LIN {X 0,Y 319.514,Z 305.497,A -85,B 0,C 180,E1 -15073.459,E2 -15073.459} C_VEL
LIN {X 0,Y 319.546,Z 305.495,A -85,B 0,C 180,E1 -15077.015,E2 -15077.015} C_VEL
LIN {X 0,Y 319.525,Z 305.485,A -85,B 0,C 180,E1 -15080.367,E2 -15080.367} C_VEL
LIN {X 0,Y 319.573,Z 305.485,A -85,B 0,C 180,E1 -15084.457,E2 -15084.457} C_VEL
LIN {X 0,Y 319.518,Z 305.495,A -85,B 0,C 180,E1 -15088.137,E2 -15088.137} C_VEL
LIN {X 0,Y 319.563,Z 305.487,A -85,B 0,C 180,E1 -15091.604,E2 -15091.604} C_VEL
LIN {X 0,Y 319.519,Z 305.494,A -85,B 0,C 180,E1 -15095.297,E2 -15095.297} C_VEL
LIN {X 0,Y 319.555,Z 305.486,A -85,B 0,C 180,E1 -15098.045,E2 -15098.045} C_VEL
LIN {X 0,Y 319.579,Z 305.489,A -85,B 0,C 180,E1 -15102.068,E2 -15102.068} C_VEL
LIN {X 0,Y 319.702,Z 305.469,A -85,B 0,C 180,E1 -15106.006,E2 -15106.006} C_VEL
LIN {X 0,Y 319.728,Z 305.469,A -85,B 0,C 180,E1 -15109.872,E2 -15109.872} C_VEL
LIN {X 0,Y 319.89,Z 305.447,A -85,B 0,C 180,E1 -15113.693,E2 -15113.693} C_VEL
LIN {X 0,Y 319.945,Z 305.439,A -85,B 0,C 180,E1 -15117.482,E2 -15117.482} C_VEL
LIN {X 0,Y 319.988,Z 305.436,A -85,B 0,C 180,E1 -15121.258,E2 -15121.258} C_VEL
LIN {X 0,Y 319.705,Z 305.464,A -85,B 0,C 180,E1 -15125.044,E2 -15125.044} C_VEL
LIN {X 0,Y 319.844,Z 305.454,A -85,B 0,C 180,E1 -15127.576,E2 -15127.576} C_VEL
LIN {X 0,Y 319.702,Z 305.473,A -85,B 0,C 180,E1 -15131.411,E2 -15131.411} C_VEL
LIN {X 0,Y 319.656,Z 305.473,A -85,B 0,C 180,E1 -15134.677,E2 -15134.677} C_VEL
LIN {X 0,Y 319.579,Z 305.489,A -85,B 0,C 180,E1 -15137.931,E2 -15137.931} C_VEL
LIN {X 0,Y 319.555,Z 305.486,A -85,B 0,C 180,E1 -15141.955,E2 -15141.955} C_VEL
LIN {X 0,Y 319.542,Z 305.492,A -85,B 0,C 180,E1 -15146.096,E2 -15146.096} C_VEL
LIN {X 0,Y 319.534,Z 305.493,A -85,B 0,C 180,E1 -15148.939,E2 -15148.939} C_VEL
LIN {X 0,Y 319.517,Z 305.495,A -85,B 0,C 180,E1 -15151.863,E2 -15151.863} C_VEL
LIN {X 0,Y 319.572,Z 305.486,A -85,B 0,C 180,E1 -15155.543,E2 -15155.543} C_VEL
LIN {X 0,Y 319.523,Z 305.485,A -85,B 0,C 180,E1 -15159.663,E2 -15159.663} C_VEL
LIN {X 0,Y 319.513,Z 305.496,A -85,B 0,C 180,E1 -15163.46,E2 -15163.46} C_VEL
LIN {X 0,Y 319.545,Z 305.488,A -85,B 0,C 180,E1 -15167.016,E2 -15167.016} C_VEL
LIN {X 0,Y 319.541,Z 305.489,A -85,B 0,C 180,E1 -15170.371,E2 -15170.371} C_VEL
LIN {X 0,Y 319.576,Z 305.488,A -85,B 0,C 180,E1 -15174.458,E2 -15174.458} C_VEL
LIN {X 0,Y 319.521,Z 305.497,A -85,B 0,C 180,E1 -15178.138,E2 -15178.138} C_VEL
LIN {X 0,Y 319.566,Z 305.489,A -85,B 0,C 180,E1 -15181.605,E2 -15181.605} C_VEL
LIN {X 0,Y 319.634,Z 305.687,A -85,B 0,C 180,E1 -15183.913,E2 -15183.913} C_VEL
LIN {X 0,Y 321.119,Z 313.482,A -85,B 0,C 180,E1 -15186.811,E2 -15186.811} C_VEL
LIN {X 0,Y 321.518,Z 317.355,A -85,B 0,C 180,E1 -15188.186,E2 -15188.186} C_VEL
LIN {X 0,Y 321.084,Z 323.649,A -85,B 0,C 180,E1 -15190.254,E2 -15190.254} C_VEL
LIN {X 0,Y 321.598,Z 327,A -85,B 0,C 180,E1 -15190.437,E2 -15190.437} C_VEL
LIN {X 0,Y 325.831,Z 351.509,A -85,B 0,C 180,E1 -15191.261,E2 -15191.261} C_VEL
LIN {X 0,Y 325.681,Z 374.115,A -85,B 0,C 180,E1 -15191.767,E2 -15191.767} C_VEL
LIN {X 0,Y 325.184,Z 400.782,A -85,B 0,C 180,E1 -15192.388,E2 -15192.388} C_VEL
LIN {X 0,Y 324.681,Z 411.953,A -85,B 0,C 180,E1 -15192.847,E2 -15192.847} C_VEL
LIN {X 0,Y 323.933,Z 423.638,A -85,B 0,C 180,E1 -15193.618,E2 -15193.618} C_VEL
LIN {X 0,Y 323.143,Z 432.319,A -85,B 0,C 180,E1 -15194.387,E2 -15194.387} C_VEL
LIN {X 0,Y 322.282,Z 440.61,A -85,B 0,C 180,E1 -15195.315,E2 -15195.315} C_VEL
LIN {X 0,Y 321.43,Z 448.456,A -85,B 0,C 180,E1 -15196.406,E2 -15196.406} C_VEL
LIN {X 0,Y 320.573,Z 455.792,A -85,B 0,C 180,E1 -15197.658,E2 -15197.658} C_VEL
LIN {X 0,Y 319.668,Z 463.231,A -85,B 0,C 180,E1 -15199.23,E2 -15199.23} C_VEL
LIN {X 0,Y 318.847,Z 470.019,A -85,B 0,C 180,E1 -15201.124,E2 -15201.124} C_VEL
LIN {X 0,Y 318.301,Z 475.173,A -85,B 0,C 180,E1 -15203.025,E2 -15203.025} C_VEL
LIN {X 0,Y 318.001,Z 478.956,A -85,B 0,C 180,E1 -15204.928,E2 -15204.928} C_VEL
LIN {X 0,Y 317.894,Z 480.692,A -85,B 0,C 180,E1 -15206.197,E2 -15206.197} C_VEL
LIN {X 0,Y 317.77,Z 481.935,A -85,B 0,C 180,E1 -15207.465,E2 -15207.465} C_VEL
LIN {X 0,Y 317.7,Z 482.708,A -85,B 0,C 180,E1 -15208.732,E2 -15208.732} C_VEL
LIN {X 0,Y 317.677,Z 483,A -85,B 0,C 180,E1 -15210,E2 -15210} C_VEL
LIN {X 0,Y 317.7,Z 482.703,A -85,B 0,C 180,E1 -15211.268,E2 -15211.268} C_VEL
LIN {X 0,Y 317.77,Z 481.92,A -85,B 0,C 180,E1 -15212.535,E2 -15212.535} C_VEL
LIN {X 0,Y 317.893,Z 480.666,A -85,B 0,C 180,E1 -15213.803,E2 -15213.803} C_VEL
LIN {X 0,Y 318.041,Z 477.844,A -85,B 0,C 180,E1 -15215.665,E2 -15215.665} C_VEL
LIN {X 0,Y 318.312,Z 475.126,A -85,B 0,C 180,E1 -15216.975,E2 -15216.975} C_VEL
LIN {X 0,Y 318.846,Z 469.956,A -85,B 0,C 180,E1 -15218.876,E2 -15218.876} C_VEL
LIN {X 0,Y 319.665,Z 463.14,A -85,B 0,C 180,E1 -15220.77,E2 -15220.77} C_VEL
LIN {X 0,Y 320.563,Z 455.687,A -85,B 0,C 180,E1 -15222.342,E2 -15222.342} C_VEL
LIN {X 0,Y 321.411,Z 448.334,A -85,B 0,C 180,E1 -15223.595,E2 -15223.595} C_VEL
LIN {X 0,Y 322.279,Z 440.457,A -85,B 0,C 180,E1 -15224.685,E2 -15224.685} C_VEL
LIN {X 0,Y 323.17,Z 432.129,A -85,B 0,C 180,E1 -15225.612,E2 -15225.612} C_VEL
LIN {X 0,Y 324.041,Z 421.482,A -85,B 0,C 180,E1 -15226.538,E2 -15226.538} C_VEL
LIN {X 0,Y 324.762,Z 409.87,A -85,B 0,C 180,E1 -15227.229,E2 -15227.229} C_VEL
LIN {X 0,Y 325.152,Z 401.415,A -85,B 0,C 180,E1 -15227.573,E2 -15227.573} C_VEL
LIN {X 0,Y 325.626,Z 375.19,A -85,B 0,C 180,E1 -15228.191,E2 -15228.191} C_VEL
LIN {X 0,Y 325.9,Z 352.19,A -85,B 0,C 180,E1 -15228.698,E2 -15228.698} C_VEL
LIN {X 0,Y 321.555,Z 326.797,A -85,B 0,C 180,E1 -15229.548,E2 -15229.548} C_VEL
LIN {X 0,Y 321.053,Z 323.814,A -85,B 0,C 180,E1 -15229.701,E2 -15229.701} C_VEL
LIN {X 0,Y 321.433,Z 319.241,A -85,B 0,C 180,E1 -15231.147,E2 -15231.147} C_VEL
LIN {X 0,Y 321.373,Z 315.374,A -85,B 0,C 180,E1 -15232.487,E2 -15232.487} C_VEL
LIN {X 0,Y 319.816,Z 306.575,A -85,B 0,C 180,E1 -15235.713,E2 -15235.713} C_VEL
LIN {X 0,Y 319.63,Z 305.559,A -85,B 0,C 180,E1 -15236.176,E2 -15236.176} C_VEL
LIN {X 0,Y 319.557,Z 305.488,A -85,B 0,C 180,E1 -15240.386,E2 -15240.386} C_VEL
LIN {X 0,Y 319.574,Z 305.491,A -85,B 0,C 180,E1 -15243.352,E2 -15243.352} C_VEL
LIN {X 0,Y 319.552,Z 305.489,A -85,B 0,C 180,E1 -15246.427,E2 -15246.427} C_VEL
LIN {X 0,Y 319.524,Z 305.491,A -85,B 0,C 180,E1 -15249.661,E2 -15249.661} C_VEL
LIN {X 0,Y 319.513,Z 305.497,A -85,B 0,C 180,E1 -15253.459,E2 -15253.459} C_VEL
LIN {X 0,Y 319.544,Z 305.495,A -85,B 0,C 180,E1 -15257.015,E2 -15257.015} C_VEL
LIN {X 0,Y 319.509,Z 305.486,A -85,B 0,C 180,E1 -15260.365,E2 -15260.365} C_VEL
LIN {X 0,Y 319.572,Z 305.486,A -85,B 0,C 180,E1 -15264.457,E2 -15264.457} C_VEL
LIN {X 0,Y 319.517,Z 305.495,A -85,B 0,C 180,E1 -15268.137,E2 -15268.137} C_VEL
LIN {X 0,Y 319.562,Z 305.487,A -85,B 0,C 180,E1 -15271.604,E2 -15271.604} C_VEL
LIN {X 0,Y 319.518,Z 305.494,A -85,B 0,C 180,E1 -15275.297,E2 -15275.297} C_VEL
LIN {X 0,Y 319.555,Z 305.486,A -85,B 0,C 180,E1 -15278.045,E2 -15278.045} C_VEL
LIN {X 0,Y 319.578,Z 305.489,A -85,B 0,C 180,E1 -15282.069,E2 -15282.069} C_VEL
LIN {X 0,Y 319.702,Z 305.469,A -85,B 0,C 180,E1 -15286.007,E2 -15286.007} C_VEL
LIN {X 0,Y 319.727,Z 305.469,A -85,B 0,C 180,E1 -15289.872,E2 -15289.872} C_VEL
LIN {X 0,Y 319.89,Z 305.447,A -85,B 0,C 180,E1 -15293.693,E2 -15293.693} C_VEL
LIN {X 0,Y 319.945,Z 305.439,A -85,B 0,C 180,E1 -15297.482,E2 -15297.482} C_VEL
LIN {X 0,Y 319.988,Z 305.436,A -85,B 0,C 180,E1 -15301.259,E2 -15301.259} C_VEL
LIN {X 0,Y 319.706,Z 305.464,A -85,B 0,C 180,E1 -15305.045,E2 -15305.045} C_VEL
LIN {X 0,Y 319.844,Z 305.454,A -85,B 0,C 180,E1 -15307.576,E2 -15307.576} C_VEL
LIN {X 0,Y 319.702,Z 305.473,A -85,B 0,C 180,E1 -15311.411,E2 -15311.411} C_VEL
LIN {X 0,Y 319.656,Z 305.473,A -85,B 0,C 180,E1 -15314.678,E2 -15314.678} C_VEL
LIN {X 0,Y 319.579,Z 305.489,A -85,B 0,C 180,E1 -15317.932,E2 -15317.932} C_VEL
LIN {X 0,Y 319.555,Z 305.486,A -85,B 0,C 180,E1 -15321.955,E2 -15321.955} C_VEL
LIN {X 0,Y 319.542,Z 305.492,A -85,B 0,C 180,E1 -15326.096,E2 -15326.096} C_VEL
LIN {X 0,Y 319.534,Z 305.493,A -85,B 0,C 180,E1 -15328.939,E2 -15328.939} C_VEL
LIN {X 0,Y 319.518,Z 305.495,A -85,B 0,C 180,E1 -15331.864,E2 -15331.864} C_VEL
LIN {X 0,Y 319.572,Z 305.486,A -85,B 0,C 180,E1 -15335.543,E2 -15335.543} C_VEL
LIN {X 0,Y 319.524,Z 305.484,A -85,B 0,C 180,E1 -15339.663,E2 -15339.663} C_VEL
LIN {X 0,Y 319.514,Z 305.496,A -85,B 0,C 180,E1 -15343.461,E2 -15343.461} C_VEL
LIN {X 0,Y 319.546,Z 305.489,A -85,B 0,C 180,E1 -15347.016,E2 -15347.016} C_VEL
LIN {X 0,Y 319.542,Z 305.488,A -85,B 0,C 180,E1 -15350.371,E2 -15350.371} C_VEL
LIN {X 0,Y 319.577,Z 305.488,A -85,B 0,C 180,E1 -15354.458,E2 -15354.458} C_VEL
LIN {X 0,Y 319.522,Z 305.496,A -85,B 0,C 180,E1 -15358.138,E2 -15358.138} C_VEL
LIN {X 0,Y 319.542,Z 305.493,A -85,B 0,C 180,E1 -15361.614,E2 -15361.614} C_VEL
LIN {X 0,Y 319.63,Z 305.684,A -85,B 0,C 180,E1 -15363.98,E2 -15363.98} C_VEL
LIN {X 0,Y 321.085,Z 313.335,A -85,B 0,C 180,E1 -15366.825,E2 -15366.825} C_VEL
LIN {X 0,Y 321.51,Z 317.158,A -85,B 0,C 180,E1 -15368.186,E2 -15368.186} C_VEL
LIN {X 0,Y 321.053,Z 323.63,A -85,B 0,C 180,E1 -15370.308,E2 -15370.308} C_VEL
LIN {X 0,Y 321.428,Z 326.151,A -85,B 0,C 180,E1 -15370.474,E2 -15370.474} C_VEL
LIN {X 0,Y 325.861,Z 352.125,A -85,B 0,C 180,E1 -15371.343,E2 -15371.343} C_VEL
LIN {X 0,Y 325.2,Z 399.977,A -85,B 0,C 180,E1 -15372.43,E2 -15372.43} C_VEL
LIN {X 0,Y 324.814,Z 408.948,A -85,B 0,C 180,E1 -15372.774,E2 -15372.774} C_VEL
LIN {X 0,Y 324.273,Z 418.484,A -85,B 0,C 180,E1 -15373.312,E2 -15373.312} C_VEL
LIN {X 0,Y 323.521,Z 428.497,A -85,B 0,C 180,E1 -15374.083,E2 -15374.083} C_VEL
LIN {X 0,Y 322.486,Z 438.884,A -85,B 0,C 180,E1 -15375.163,E2 -15375.163} C_VEL
LIN {X 0,Y 321.565,Z 447.028,A -85,B 0,C 180,E1 -15376.251,E2 -15376.251} C_VEL
LIN {X 0,Y 320.834,Z 453.747,A -85,B 0,C 180,E1 -15377.347,E2 -15377.347} C_VEL
LIN {X 0,Y 320.021,Z 460.112,A -85,B 0,C 180,E1 -15378.601,E2 -15378.601} C_VEL
LIN {X 0,Y 319.24,Z 466.576,A -85,B 0,C 180,E1 -15380.177,E2 -15380.177} C_VEL
LIN {X 0,Y 318.679,Z 471.734,A -85,B 0,C 180,E1 -15381.759,E2 -15381.759} C_VEL
LIN {X 0,Y 318.157,Z 476.676,A -85,B 0,C 180,E1 -15383.741,E2 -15383.741} C_VEL
LIN {X 0,Y 318.009,Z 478.838,A -85,B 0,C 180,E1 -15384.929,E2 -15384.929} C_VEL
LIN {X 0,Y 317.899,Z 480.609,A -85,B 0,C 180,E1 -15386.197,E2 -15386.197} C_VEL
LIN {X 0,Y 317.772,Z 481.886,A -85,B 0,C 180,E1 -15387.465,E2 -15387.465} C_VEL
LIN {X 0,Y 317.701,Z 482.691,A -85,B 0,C 180,E1 -15388.732,E2 -15388.732} C_VEL
LIN {X 0,Y 317.679,Z 482.998,A -85,B 0,C 180,E1 -15390,E2 -15390} C_VEL
LIN {X 0,Y 317.697,Z 482.719,A -85,B 0,C 180,E1 -15391.268,E2 -15391.268} C_VEL
LIN {X 0,Y 317.76,Z 481.97,A -85,B 0,C 180,E1 -15392.535,E2 -15392.535} C_VEL
LIN {X 0,Y 317.87,Z 480.75,A -85,B 0,C 180,E1 -15393.803,E2 -15393.803} C_VEL
LIN {X 0,Y 318.029,Z 478.009,A -85,B 0,C 180,E1 -15395.639,E2 -15395.639} C_VEL
LIN {X 0,Y 318.309,Z 475.28,A -85,B 0,C 180,E1 -15396.975,E2 -15396.975} C_VEL
LIN {X 0,Y 318.839,Z 470.153,A -85,B 0,C 180,E1 -15398.876,E2 -15398.876} C_VEL
LIN {X 0,Y 319.502,Z 464.639,A -85,B 0,C 180,E1 -15400.455,E2 -15400.455} C_VEL
LIN {X 0,Y 320.377,Z 457.713,A -85,B 0,C 180,E1 -15402.028,E2 -15402.028} C_VEL
LIN {X 0,Y 321.284,Z 449.762,A -85,B 0,C 180,E1 -15403.439,E2 -15403.439} C_VEL
LIN {X 0,Y 322.108,Z 442.181,A -85,B 0,C 180,E1 -15404.531,E2 -15404.531} C_VEL
LIN {X 0,Y 323.005,Z 434.237,A -85,B 0,C 180,E1 -15405.458,E2 -15405.458} C_VEL
LIN {X 0,Y 323.747,Z 426.031,A -85,B 0,C 180,E1 -15406.23,E2 -15406.23} C_VEL
LIN {X 0,Y 324.389,Z 417.714,A -85,B 0,C 180,E1 -15406.844,E2 -15406.844} C_VEL
LIN {X 0,Y 324.828,Z 408.722,A -85,B 0,C 180,E1 -15407.347,E2 -15407.347} C_VEL
LIN {X 0,Y 325.258,Z 399.317,A -85,B 0,C 180,E1 -15407.699,E2 -15407.699} C_VEL
LIN {X 0,Y 325.92,Z 352.078,A -85,B 0,C 180,E1 -15408.765,E2 -15408.765} C_VEL
LIN {X 0,Y 321.836,Z 328.161,A -85,B 0,C 180,E1 -15409.566,E2 -15409.566} C_VEL
LIN {X 0,Y 321.058,Z 323.761,A -85,B 0,C 180,E1 -15409.776,E2 -15409.776} C_VEL
LIN {X 0,Y 321.492,Z 317.485,A -85,B 0,C 180,E1 -15411.816,E2 -15411.816} C_VEL
LIN {X 0,Y 320.766,Z 311.628,A -85,B 0,C 180,E1 -15413.912,E2 -15413.912} C_VEL
LIN {X 0,Y 319.606,Z 305.566,A -85,B 0,C 180,E1 -15416.222,E2 -15416.222} C_VEL
LIN {X 0,Y 319.541,Z 305.493,A -85,B 0,C 180,E1 -15418.938,E2 -15418.938} C_VEL
LIN {X 0,Y 319.522,Z 305.497,A -85,B 0,C 180,E1 -15421.862,E2 -15421.862} C_VEL
LIN {X 0,Y 319.577,Z 305.487,A -85,B 0,C 180,E1 -15425.542,E2 -15425.542} C_VEL
LIN {X 0,Y 319.525,Z 305.491,A -85,B 0,C 180,E1 -15429.661,E2 -15429.661} C_VEL
LIN {X 0,Y 319.491,Z 305.492,A -85,B 0,C 180,E1 -15431.235,E2 -15431.235} C_VEL
LIN {X 0,Y 318.864,Z 305.576,A -85,B 0,C 180,E1 -15432.287,E2 -15432.287} C_VEL
LIN {X 0,Y 316.003,Z 305.934,A -85,B 0,C 180,E1 -15433.997,E2 -15433.997} C_VEL
LIN {X 0,Y 313.554,Z 306.241,A -85,B 0,C 180,E1 -15435.383,E2 -15435.383} C_VEL
LIN {X 0,Y 312.509,Z 306.368,A -85,B 0,C 180,E1 -15436.458,E2 -15436.458} C_VEL
LIN {X 0,Y 312.429,Z 306.374,A -85,B 0,C 180,E1 -15436.822,E2 -15436.822} C_VEL
LIN {X 0,Y 312.46,Z 306.361,A -85,B 0,C 180,E1 -15440.965,E2 -15440.965} C_VEL
LIN {X 0,Y 312.524,Z 306.362,A -85,B 0,C 180,E1 -15444.219,E2 -15444.219} C_VEL
LIN {X 0,Y 312.496,Z 306.37,A -85,B 0,C 180,E1 -15447.333,E2 -15447.333} C_VEL
LIN {X 0,Y 312.498,Z 306.368,A -85,B 0,C 180,E1 -15451.292,E2 -15451.292} C_VEL
LIN {X 0,Y 312.51,Z 306.371,A -85,B 0,C 180,E1 -15454.704,E2 -15454.704} C_VEL
LIN {X 0,Y 312.532,Z 306.359,A -85,B 0,C 180,E1 -15457.525,E2 -15457.525} C_VEL
LIN {X 0,Y 312.539,Z 306.364,A -85,B 0,C 180,E1 -15461.65,E2 -15461.65} C_VEL
LIN {X 0,Y 312.644,Z 306.346,A -85,B 0,C 180,E1 -15465.684,E2 -15465.684} C_VEL
LIN {X 0,Y 312.678,Z 306.346,A -85,B 0,C 180,E1 -15469.641,E2 -15469.641} C_VEL
LIN {X 0,Y 312.788,Z 306.335,A -85,B 0,C 180,E1 -15472.252,E2 -15472.252} C_VEL
LIN {X 0,Y 312.677,Z 306.339,A -85,B 0,C 180,E1 -15474.842,E2 -15474.842} C_VEL
LIN {X 0,Y 312.957,Z 306.312,A -85,B 0,C 180,E1 -15478.713,E2 -15478.713} C_VEL
LIN {X 0,Y 312.956,Z 306.312,A -85,B 0,C 180,E1 -15481.287,E2 -15481.287} C_VEL
LIN {X 0,Y 312.832,Z 306.326,A -85,B 0,C 180,E1 -15486.449,E2 -15486.449} C_VEL
LIN {X 0,Y 312.675,Z 306.346,A -85,B 0,C 180,E1 -15490.359,E2 -15490.359} C_VEL
LIN {X 0,Y 312.643,Z 306.346,A -85,B 0,C 180,E1 -15494.316,E2 -15494.316} C_VEL
LIN {X 0,Y 312.539,Z 306.364,A -85,B 0,C 180,E1 -15498.35,E2 -15498.35} C_VEL
LIN {X 0,Y 312.531,Z 306.359,A -85,B 0,C 180,E1 -15502.475,E2 -15502.475} C_VEL
LIN {X 0,Y 312.5,Z 306.37,A -85,B 0,C 180,E1 -15505.899,E2 -15505.899} C_VEL
LIN {X 0,Y 312.488,Z 306.368,A -85,B 0,C 180,E1 -15509.656,E2 -15509.656} C_VEL
LIN {X 0,Y 312.513,Z 306.368,A -85,B 0,C 180,E1 -15513.689,E2 -15513.689} C_VEL
LIN {X 0,Y 312.503,Z 306.359,A -85,B 0,C 180,E1 -15517.388,E2 -15517.388} C_VEL
LIN {X 0,Y 312.435,Z 306.368,A -85,B 0,C 180,E1 -15520.718,E2 -15520.718} C_VEL
LIN {X 0,Y 312.444,Z 306.376,A -85,B 0,C 180,E1 -15524.211,E2 -15524.211} C_VEL
LIN {X 0,Y 312.448,Z 306.367,A -85,B 0,C 180,E1 -15527.926,E2 -15527.926} C_VEL
LIN {X 0,Y 312.479,Z 306.372,A -85,B 0,C 180,E1 -15531.923,E2 -15531.923} C_VEL
LIN {X 0,Y 312.527,Z 306.366,A -85,B 0,C 180,E1 -15534.221,E2 -15534.221} C_VEL
LIN {X 0,Y 312.498,Z 306.37,A -85,B 0,C 180,E1 -15537.334,E2 -15537.334} C_VEL
LIN {X 0,Y 312.502,Z 306.369,A -85,B 0,C 180,E1 -15541.293,E2 -15541.293} C_VEL
LIN {X 0,Y 312.588,Z 306.579,A -85,B 0,C 180,E1 -15543.61,E2 -15543.61} C_VEL
LIN {X 0,Y 314.303,Z 315.843,A -85,B 0,C 180,E1 -15547.121,E2 -15547.121} C_VEL
LIN {X 0,Y 314.384,Z 321.26,A -85,B 0,C 180,E1 -15549.043,E2 -15549.043} C_VEL
LIN {X 0,Y 314.178,Z 323.787,A -85,B 0,C 180,E1 -15549.822,E2 -15549.822} C_VEL
LIN {X 0,Y 315.376,Z 330.306,A -85,B 0,C 180,E1 -15550.113,E2 -15550.113} C_VEL
LIN {X 0,Y 319.287,Z 353.525,A -85,B 0,C 180,E1 -15550.909,E2 -15550.909} C_VEL
LIN {X 0,Y 318.496,Z 399.599,A -85,B 0,C 180,E1 -15551.967,E2 -15551.967} C_VEL
LIN {X 0,Y 318.075,Z 408.641,A -85,B 0,C 180,E1 -15552.314,E2 -15552.314} C_VEL
LIN {X 0,Y 317.489,Z 418.259,A -85,B 0,C 180,E1 -15552.862,E2 -15552.862} C_VEL
LIN {X 0,Y 316.805,Z 427.389,A -85,B 0,C 180,E1 -15553.57,E2 -15553.57} C_VEL
LIN {X 0,Y 315.736,Z 438.154,A -85,B 0,C 180,E1 -15554.673,E2 -15554.673} C_VEL
LIN {X 0,Y 314.752,Z 446.418,A -85,B 0,C 180,E1 -15555.782,E2 -15555.782} C_VEL
LIN {X 0,Y 313.854,Z 454.091,A -85,B 0,C 180,E1 -15557.061,E2 -15557.061} C_VEL
LIN {X 0,Y 313.039,Z 460.404,A -85,B 0,C 180,E1 -15558.343,E2 -15558.343} C_VEL
LIN {X 0,Y 312.335,Z 465.648,A -85,B 0,C 180,E1 -15559.63,E2 -15559.63} C_VEL
LIN {X 0,Y 311.818,Z 470.02,A -85,B 0,C 180,E1 -15560.923,E2 -15560.923} C_VEL
LIN {X 0,Y 311.246,Z 475.174,A -85,B 0,C 180,E1 -15562.866,E2 -15562.866} C_VEL
LIN {X 0,Y 310.916,Z 478.956,A -85,B 0,C 180,E1 -15564.813,E2 -15564.813} C_VEL
LIN {X 0,Y 310.809,Z 480.693,A -85,B 0,C 180,E1 -15566.11,E2 -15566.11} C_VEL
LIN {X 0,Y 310.696,Z 481.936,A -85,B 0,C 180,E1 -15567.407,E2 -15567.407} C_VEL
LIN {X 0,Y 310.617,Z 482.708,A -85,B 0,C 180,E1 -15568.704,E2 -15568.704} C_VEL
LIN {X 0,Y 310.592,Z 483,A -85,B 0,C 180,E1 -15570,E2 -15570} C_VEL
LIN {X 0,Y 310.617,Z 482.703,A -85,B 0,C 180,E1 -15571.296,E2 -15571.296} C_VEL
LIN {X 0,Y 310.696,Z 481.92,A -85,B 0,C 180,E1 -15572.593,E2 -15572.593} C_VEL
LIN {X 0,Y 310.808,Z 480.666,A -85,B 0,C 180,E1 -15573.89,E2 -15573.89} C_VEL
LIN {X 0,Y 310.912,Z 478.918,A -85,B 0,C 180,E1 -15575.188,E2 -15575.188} C_VEL
LIN {X 0,Y 311.251,Z 475.125,A -85,B 0,C 180,E1 -15577.134,E2 -15577.134} C_VEL
LIN {X 0,Y 311.817,Z 469.955,A -85,B 0,C 180,E1 -15579.077,E2 -15579.077} C_VEL
LIN {X 0,Y 312.667,Z 463.138,A -85,B 0,C 180,E1 -15581.014,E2 -15581.014} C_VEL
LIN {X 0,Y 313.64,Z 455.684,A -85,B 0,C 180,E1 -15582.619,E2 -15582.619} C_VEL
LIN {X 0,Y 314.501,Z 448.331,A -85,B 0,C 180,E1 -15583.899,E2 -15583.899} C_VEL
LIN {X 0,Y 315.434,Z 440.453,A -85,B 0,C 180,E1 -15585.011,E2 -15585.011} C_VEL
LIN {X 0,Y 316.354,Z 432.124,A -85,B 0,C 180,E1 -15585.957,E2 -15585.957} C_VEL
LIN {X 0,Y 317.24,Z 421.476,A -85,B 0,C 180,E1 -15586.903,E2 -15586.903} C_VEL
LIN {X 0,Y 318.004,Z 409.861,A -85,B 0,C 180,E1 -15587.607,E2 -15587.607} C_VEL
LIN {X 0,Y 318.41,Z 401.4,A -85,B 0,C 180,E1 -15587.958,E2 -15587.958} C_VEL
LIN {X 0,Y 318.889,Z 375.169,A -85,B 0,C 180,E1 -15588.589,E2 -15588.589} C_VEL
LIN {X 0,Y 319.191,Z 353.155,A -85,B 0,C 180,E1 -15589.083,E2 -15589.083} C_VEL
LIN {X 0,Y 314.775,Z 327.23,A -85,B 0,C 180,E1 -15589.976,E2 -15589.976} C_VEL
LIN {X 0,Y 314.159,Z 323.735,A -85,B 0,C 180,E1 -15590.165,E2 -15590.165} C_VEL
LIN {X 0,Y 314.491,Z 319.239,A -85,B 0,C 180,E1 -15591.637,E2 -15591.637} C_VEL
LIN {X 0,Y 314.047,Z 314.28,A -85,B 0,C 180,E1 -15593.432,E2 -15593.432} C_VEL
LIN {X 0,Y 312.57,Z 306.452,A -85,B 0,C 180,E1 -15596.446,E2 -15596.446} C_VEL
LIN {X 0,Y 312.493,Z 306.372,A -85,B 0,C 180,E1 -15599.655,E2 -15599.655} C_VEL
LIN {X 0,Y 312.517,Z 306.366,A -85,B 0,C 180,E1 -15603.688,E2 -15603.688} C_VEL
LIN {X 0,Y 312.51,Z 306.372,A -85,B 0,C 180,E1 -15607.386,E2 -15607.386} C_VEL
LIN {X 0,Y 312.435,Z 306.372,A -85,B 0,C 180,E1 -15610.717,E2 -15610.717} C_VEL
LIN {X 0,Y 312.445,Z 306.374,A -85,B 0,C 180,E1 -15614.21,E2 -15614.21} C_VEL
LIN {X 0,Y 312.448,Z 306.372,A -85,B 0,C 180,E1 -15617.925,E2 -15617.925} C_VEL
LIN {X 0,Y 312.469,Z 306.361,A -85,B 0,C 180,E1 -15621.924,E2 -15621.924} C_VEL
LIN {X 0,Y 312.523,Z 306.362,A -85,B 0,C 180,E1 -15624.219,E2 -15624.219} C_VEL
LIN {X 0,Y 312.495,Z 306.37,A -85,B 0,C 180,E1 -15627.333,E2 -15627.333} C_VEL
LIN {X 0,Y 312.498,Z 306.368,A -85,B 0,C 180,E1 -15631.292,E2 -15631.292} C_VEL
LIN {X 0,Y 312.509,Z 306.371,A -85,B 0,C 180,E1 -15634.704,E2 -15634.704} C_VEL
LIN {X 0,Y 312.531,Z 306.359,A -85,B 0,C 180,E1 -15637.525,E2 -15637.525} C_VEL
LIN {X 0,Y 312.539,Z 306.364,A -85,B 0,C 180,E1 -15641.65,E2 -15641.65} C_VEL
LIN {X 0,Y 312.644,Z 306.346,A -85,B 0,C 180,E1 -15645.684,E2 -15645.684} C_VEL
LIN {X 0,Y 312.677,Z 306.346,A -85,B 0,C 180,E1 -15649.641,E2 -15649.641} C_VEL
LIN {X 0,Y 312.788,Z 306.335,A -85,B 0,C 180,E1 -15652.252,E2 -15652.252} C_VEL
LIN {X 0,Y 312.677,Z 306.339,A -85,B 0,C 180,E1 -15654.842,E2 -15654.842} C_VEL
LIN {X 0,Y 312.957,Z 306.312,A -85,B 0,C 180,E1 -15658.713,E2 -15658.713} C_VEL
LIN {X 0,Y 312.956,Z 306.312,A -85,B 0,C 180,E1 -15661.287,E2 -15661.287} C_VEL
LIN {X 0,Y 312.832,Z 306.325,A -85,B 0,C 180,E1 -15666.45,E2 -15666.45} C_VEL
LIN {X 0,Y 312.675,Z 306.346,A -85,B 0,C 180,E1 -15670.359,E2 -15670.359} C_VEL
LIN {X 0,Y 312.644,Z 306.346,A -85,B 0,C 180,E1 -15674.316,E2 -15674.316} C_VEL
LIN {X 0,Y 312.539,Z 306.364,A -85,B 0,C 180,E1 -15678.35,E2 -15678.35} C_VEL
LIN {X 0,Y 312.532,Z 306.358,A -85,B 0,C 180,E1 -15682.475,E2 -15682.475} C_VEL
LIN {X 0,Y 312.5,Z 306.37,A -85,B 0,C 180,E1 -15685.899,E2 -15685.899} C_VEL
LIN {X 0,Y 312.488,Z 306.368,A -85,B 0,C 180,E1 -15689.656,E2 -15689.656} C_VEL
LIN {X 0,Y 312.514,Z 306.368,A -85,B 0,C 180,E1 -15693.689,E2 -15693.689} C_VEL
LIN {X 0,Y 312.504,Z 306.359,A -85,B 0,C 180,E1 -15697.388,E2 -15697.388} C_VEL
LIN {X 0,Y 312.436,Z 306.367,A -85,B 0,C 180,E1 -15700.718,E2 -15700.718} C_VEL
LIN {X 0,Y 312.446,Z 306.376,A -85,B 0,C 180,E1 -15704.211,E2 -15704.211} C_VEL
LIN {X 0,Y 312.449,Z 306.367,A -85,B 0,C 180,E1 -15707.926,E2 -15707.926} C_VEL
LIN {X 0,Y 312.481,Z 306.371,A -85,B 0,C 180,E1 -15711.923,E2 -15711.923} C_VEL
LIN {X 0,Y 312.528,Z 306.365,A -85,B 0,C 180,E1 -15714.221,E2 -15714.221} C_VEL
LIN {X 0,Y 312.499,Z 306.37,A -85,B 0,C 180,E1 -15717.334,E2 -15717.334} C_VEL
LIN {X 0,Y 312.482,Z 306.373,A -85,B 0,C 180,E1 -15721.3,E2 -15721.3} C_VEL
LIN {X 0,Y 312.565,Z 306.569,A -85,B 0,C 180,E1 -15723.672,E2 -15723.672} C_VEL
LIN {X 0,Y 314.046,Z 314.156,A -85,B 0,C 180,E1 -15726.568,E2 -15726.568} C_VEL
LIN {X 0,Y 314.49,Z 319.112,A -85,B 0,C 180,E1 -15728.363,E2 -15728.363} C_VEL
LIN {X 0,Y 314.195,Z 323.825,A -85,B 0,C 180,E1 -15729.897,E2 -15729.897} C_VEL
LIN {X 0,Y 315.548,Z 331.299,A -85,B 0,C 180,E1 -15730.216,E2 -15730.216} C_VEL
LIN {X 0,Y 319.258,Z 353.736,A -85,B 0,C 180,E1 -15730.98,E2 -15730.98} C_VEL
LIN {X 0,Y 318.433,Z 399.995,A -85,B 0,C 180,E1 -15732.044,E2 -15732.044} C_VEL
LIN {X 0,Y 318.015,Z 409.791,A -85,B 0,C 180,E1 -15732.435,E2 -15732.435} C_VEL
LIN {X 0,Y 317.329,Z 420.889,A -85,B 0,C 180,E1 -15733.101,E2 -15733.101} C_VEL
LIN {X 0,Y 316.352,Z 431.716,A -85,B 0,C 180,E1 -15734.043,E2 -15734.043} C_VEL
LIN {X 0,Y 315.483,Z 440.118,A -85,B 0,C 180,E1 -15734.991,E2 -15734.991} C_VEL
LIN {X 0,Y 314.679,Z 447.031,A -85,B 0,C 180,E1 -15735.944,E2 -15735.944} C_VEL
LIN {X 0,Y 313.897,Z 453.75,A -85,B 0,C 180,E1 -15737.062,E2 -15737.062} C_VEL
LIN {X 0,Y 313.051,Z 460.114,A -85,B 0,C 180,E1 -15738.343,E2 -15738.343} C_VEL
LIN {X 0,Y 312.245,Z 466.578,A -85,B 0,C 180,E1 -15739.954,E2 -15739.954} C_VEL
LIN {X 0,Y 311.657,Z 471.736,A -85,B 0,C 180,E1 -15741.572,E2 -15741.572} C_VEL
LIN {X 0,Y 311.111,Z 476.509,A -85,B 0,C 180,E1 -15743.515,E2 -15743.515} C_VEL
LIN {X 0,Y 310.923,Z 478.839,A -85,B 0,C 180,E1 -15744.813,E2 -15744.813} C_VEL
LIN {X 0,Y 310.814,Z 480.61,A -85,B 0,C 180,E1 -15746.11,E2 -15746.11} C_VEL
LIN {X 0,Y 310.698,Z 481.886,A -85,B 0,C 180,E1 -15747.407,E2 -15747.407} C_VEL
LIN {X 0,Y 310.619,Z 482.692,A -85,B 0,C 180,E1 -15748.704,E2 -15748.704} C_VEL
LIN {X 0,Y 310.593,Z 482.998,A -85,B 0,C 180,E1 -15750,E2 -15750} C_VEL
LIN {X 0,Y 310.615,Z 482.719,A -85,B 0,C 180,E1 -15751.296,E2 -15751.296} C_VEL
LIN {X 0,Y 310.686,Z 481.969,A -85,B 0,C 180,E1 -15752.593,E2 -15752.593} C_VEL
LIN {X 0,Y 310.787,Z 480.749,A -85,B 0,C 180,E1 -15753.89,E2 -15753.89} C_VEL
LIN {X 0,Y 310.907,Z 479.036,A -85,B 0,C 180,E1 -15755.188,E2 -15755.188} C_VEL
LIN {X 0,Y 311.25,Z 475.279,A -85,B 0,C 180,E1 -15757.134,E2 -15757.134} C_VEL
LIN {X 0,Y 311.807,Z 470.152,A -85,B 0,C 180,E1 -15759.078,E2 -15759.078} C_VEL
LIN {X 0,Y 312.53,Z 464.637,A -85,B 0,C 180,E1 -15760.691,E2 -15760.691} C_VEL
LIN {X 0,Y 313.412,Z 457.71,A -85,B 0,C 180,E1 -15762.3,E2 -15762.3} C_VEL
LIN {X 0,Y 314.375,Z 449.758,A -85,B 0,C 180,E1 -15763.74,E2 -15763.74} C_VEL
LIN {X 0,Y 315.258,Z 442.177,A -85,B 0,C 180,E1 -15764.854,E2 -15764.854} C_VEL
LIN {X 0,Y 316.178,Z 434.232,A -85,B 0,C 180,E1 -15765.8,E2 -15765.8} C_VEL
LIN {X 0,Y 316.937,Z 426.025,A -85,B 0,C 180,E1 -15766.588,E2 -15766.588} C_VEL
LIN {X 0,Y 317.616,Z 417.706,A -85,B 0,C 180,E1 -15767.214,E2 -15767.214} C_VEL
LIN {X 0,Y 318.072,Z 408.71,A -85,B 0,C 180,E1 -15767.728,E2 -15767.728} C_VEL
LIN {X 0,Y 318.487,Z 399.774,A -85,B 0,C 180,E1 -15768.072,E2 -15768.072} C_VEL
LIN {X 0,Y 319.254,Z 353.243,A -85,B 0,C 180,E1 -15769.145,E2 -15769.145} C_VEL
LIN {X 0,Y 315.148,Z 329.211,A -85,B 0,C 180,E1 -15769.973,E2 -15769.973} C_VEL
LIN {X 0,Y 314.179,Z 323.787,A -85,B 0,C 180,E1 -15770.223,E2 -15770.223} C_VEL
LIN {X 0,Y 314.477,Z 319.436,A -85,B 0,C 180,E1 -15771.638,E2 -15771.638} C_VEL
LIN {X 0,Y 314.066,Z 314.451,A -85,B 0,C 180,E1 -15773.44,E2 -15773.44} C_VEL
LIN {X 0,Y 312.576,Z 306.464,A -85,B 0,C 180,E1 -15776.503,E2 -15776.503} C_VEL
LIN {X 0,Y 312.494,Z 306.372,A -85,B 0,C 180,E1 -15779.655,E2 -15779.655} C_VEL
LIN {X 0,Y 312.518,Z 306.366,A -85,B 0,C 180,E1 -15783.688,E2 -15783.688} C_VEL
LIN {X 0,Y 312.511,Z 306.372,A -85,B 0,C 180,E1 -15787.386,E2 -15787.386} C_VEL
LIN {X 0,Y 312.421,Z 306.37,A -85,B 0,C 180,E1 -15791.234,E2 -15791.234} C_VEL
LIN {X 0,Y 312.446,Z 306.374,A -85,B 0,C 180,E1 -15794.209,E2 -15794.209} C_VEL
LIN {X 0,Y 312.429,Z 306.374,A -85,B 0,C 180,E1 -15796.822,E2 -15796.822} C_VEL
LIN {X 0,Y 311.773,Z 306.458,A -85,B 0,C 180,E1 -15797.897,E2 -15797.897} C_VEL
LIN {X 0,Y 308.924,Z 306.803,A -85,B 0,C 180,E1 -15799.647,E2 -15799.647} C_VEL
LIN {X 0,Y 306.511,Z 307.1,A -85,B 0,C 180,E1 -15801.066,E2 -15801.066} C_VEL
LIN {X 0,Y 305.488,Z 307.228,A -85,B 0,C 180,E1 -15802.166,E2 -15802.166} C_VEL
LIN {X 0,Y 305.412,Z 307.239,A -85,B 0,C 180,E1 -15802.538,E2 -15802.538} C_VEL
LIN {X 0,Y 305.46,Z 307.247,A -85,B 0,C 180,E1 -15806.482,E2 -15806.482} C_VEL
LIN {X 0,Y 305.424,Z 307.246,A -85,B 0,C 180,E1 -15809.586,E2 -15809.586} C_VEL
LIN {X 0,Y 305.443,Z 307.25,A -85,B 0,C 180,E1 -15812.601,E2 -15812.601} C_VEL
LIN {X 0,Y 305.433,Z 307.248,A -85,B 0,C 180,E1 -15815.532,E2 -15815.532} C_VEL
LIN {X 0,Y 305.469,Z 307.242,A -85,B 0,C 180,E1 -15819.811,E2 -15819.811} C_VEL
LIN {X 0,Y 305.506,Z 307.24,A -85,B 0,C 180,E1 -15823.975,E2 -15823.975} C_VEL
LIN {X 0,Y 305.563,Z 307.229,A -85,B 0,C 180,E1 -15826.703,E2 -15826.703} C_VEL
LIN {X 0,Y 305.746,Z 307.209,A -85,B 0,C 180,E1 -15831.261,E2 -15831.261} C_VEL
LIN {X 0,Y 305.777,Z 307.203,A -85,B 0,C 180,E1 -15833.401,E2 -15833.401} C_VEL
LIN {X 0,Y 305.926,Z 307.188,A -85,B 0,C 180,E1 -15838.683,E2 -15838.683} C_VEL
LIN {X 0,Y 305.925,Z 307.188,A -85,B 0,C 180,E1 -15841.316,E2 -15841.316} C_VEL
LIN {X 0,Y 305.777,Z 307.203,A -85,B 0,C 180,E1 -15846.599,E2 -15846.599} C_VEL
LIN {X 0,Y 305.676,Z 307.219,A -85,B 0,C 180,E1 -15849.261,E2 -15849.261} C_VEL
LIN {X 0,Y 305.561,Z 307.229,A -85,B 0,C 180,E1 -15853.297,E2 -15853.297} C_VEL
LIN {X 0,Y 305.506,Z 307.241,A -85,B 0,C 180,E1 -15856.025,E2 -15856.025} C_VEL
LIN {X 0,Y 305.469,Z 307.242,A -85,B 0,C 180,E1 -15860.188,E2 -15860.188} C_VEL
LIN {X 0,Y 305.432,Z 307.248,A -85,B 0,C 180,E1 -15864.468,E2 -15864.468} C_VEL
LIN {X 0,Y 305.442,Z 307.25,A -85,B 0,C 180,E1 -15867.399,E2 -15867.399} C_VEL
LIN {X 0,Y 305.423,Z 307.246,A -85,B 0,C 180,E1 -15870.413,E2 -15870.413} C_VEL
LIN {X 0,Y 305.458,Z 307.245,A -85,B 0,C 180,E1 -15874.079,E2 -15874.079} C_VEL
LIN {X 0,Y 305.445,Z 307.243,A -85,B 0,C 180,E1 -15876.743,E2 -15876.743} C_VEL
LIN {X 0,Y 305.403,Z 307.242,A -85,B 0,C 180,E1 -15880.59,E2 -15880.59} C_VEL
LIN {X 0,Y 305.415,Z 307.252,A -85,B 0,C 180,E1 -15883.657,E2 -15883.657} C_VEL
LIN {X 0,Y 305.429,Z 307.241,A -85,B 0,C 180,E1 -15887.419,E2 -15887.419} C_VEL
LIN {X 0,Y 305.456,Z 307.246,A -85,B 0,C 180,E1 -15891.596,E2 -15891.596} C_VEL
LIN {X 0,Y 305.458,Z 307.242,A -85,B 0,C 180,E1 -15894.887,E2 -15894.887} C_VEL
LIN {X 0,Y 305.439,Z 307.25,A -85,B 0,C 180,E1 -15898.359,E2 -15898.359} C_VEL
LIN {X 0,Y 305.471,Z 307.246,A -85,B 0,C 180,E1 -15901.11,E2 -15901.11} C_VEL
LIN {X 0,Y 305.522,Z 307.38,A -85,B 0,C 180,E1 -15903.24,E2 -15903.24} C_VEL
LIN {X 0,Y 307.216,Z 316.266,A -85,B 0,C 180,E1 -15906.716,E2 -15906.716} C_VEL
LIN {X 0,Y 307.469,Z 321.262,A -85,B 0,C 180,E1 -15908.549,E2 -15908.549} C_VEL
LIN {X 0,Y 307.315,Z 323.971,A -85,B 0,C 180,E1 -15909.371,E2 -15909.371} C_VEL
LIN {X 0,Y 310.978,Z 344.06,A -85,B 0,C 180,E1 -15910.15,E2 -15910.15} C_VEL
LIN {X 0,Y 312.57,Z 355.106,A -85,B 0,C 180,E1 -15910.519,E2 -15910.519} C_VEL
LIN {X 0,Y 311.758,Z 399.698,A -85,B 0,C 180,E1 -15911.567,E2 -15911.567} C_VEL
LIN {X 0,Y 311.272,Z 409.482,A -85,B 0,C 180,E1 -15911.956,E2 -15911.956} C_VEL
LIN {X 0,Y 310.655,Z 419.476,A -85,B 0,C 180,E1 -15912.557,E2 -15912.557} C_VEL
LIN {X 0,Y 309.661,Z 430.827,A -85,B 0,C 180,E1 -15913.519,E2 -15913.519} C_VEL
LIN {X 0,Y 308.753,Z 439.388,A -85,B 0,C 180,E1 -15914.487,E2 -15914.487} C_VEL
LIN {X 0,Y 307.749,Z 447.442,A -85,B 0,C 180,E1 -15915.62,E2 -15915.62} C_VEL
LIN {X 0,Y 306.924,Z 454.093,A -85,B 0,C 180,E1 -15916.763,E2 -15916.763} C_VEL
LIN {X 0,Y 306.078,Z 460.406,A -85,B 0,C 180,E1 -15918.074,E2 -15918.074} C_VEL
LIN {X 0,Y 305.362,Z 465.65,A -85,B 0,C 180,E1 -15919.39,E2 -15919.39} C_VEL
LIN {X 0,Y 304.813,Z 470.022,A -85,B 0,C 180,E1 -15920.712,E2 -15920.712} C_VEL
LIN {X 0,Y 304.2,Z 475.175,A -85,B 0,C 180,E1 -15922.7,E2 -15922.7} C_VEL
LIN {X 0,Y 303.84,Z 478.957,A -85,B 0,C 180,E1 -15924.691,E2 -15924.691} C_VEL
LIN {X 0,Y 303.726,Z 480.693,A -85,B 0,C 180,E1 -15926.02,E2 -15926.02} C_VEL
LIN {X 0,Y 303.624,Z 481.936,A -85,B 0,C 180,E1 -15927.347,E2 -15927.347} C_VEL
LIN {X 0,Y 303.537,Z 482.708,A -85,B 0,C 180,E1 -15928.673,E2 -15928.673} C_VEL
LIN {X 0,Y 303.51,Z 483,A -85,B 0,C 180,E1 -15930,E2 -15930} C_VEL
LIN {X 0,Y 303.537,Z 482.703,A -85,B 0,C 180,E1 -15931.327,E2 -15931.327} C_VEL
LIN {X 0,Y 303.624,Z 481.919,A -85,B 0,C 180,E1 -15932.653,E2 -15932.653} C_VEL
LIN {X 0,Y 303.725,Z 480.665,A -85,B 0,C 180,E1 -15933.98,E2 -15933.98} C_VEL
LIN {X 0,Y 303.834,Z 478.917,A -85,B 0,C 180,E1 -15935.309,E2 -15935.309} C_VEL
LIN {X 0,Y 304.202,Z 475.124,A -85,B 0,C 180,E1 -15937.3,E2 -15937.3} C_VEL
LIN {X 0,Y 304.811,Z 469.954,A -85,B 0,C 180,E1 -15939.288,E2 -15939.288} C_VEL
LIN {X 0,Y 305.681,Z 463.136,A -85,B 0,C 180,E1 -15941.269,E2 -15941.269} C_VEL
LIN {X 0,Y 306.72,Z 455.682,A -85,B 0,C 180,E1 -15942.909,E2 -15942.909} C_VEL
LIN {X 0,Y 307.626,Z 448.328,A -85,B 0,C 180,E1 -15944.217,E2 -15944.217} C_VEL
LIN {X 0,Y 308.594,Z 440.45,A -85,B 0,C 180,E1 -15945.352,E2 -15945.352} C_VEL
LIN {X 0,Y 309.545,Z 432.12,A -85,B 0,C 180,E1 -15946.317,E2 -15946.317} C_VEL
LIN {X 0,Y 310.467,Z 421.47,A -85,B 0,C 180,E1 -15947.284,E2 -15947.284} C_VEL
LIN {X 0,Y 311.262,Z 409.851,A -85,B 0,C 180,E1 -15948.002,E2 -15948.002} C_VEL
LIN {X 0,Y 311.672,Z 401.385,A -85,B 0,C 180,E1 -15948.36,E2 -15948.36} C_VEL
LIN {X 0,Y 312.185,Z 374.532,A -85,B 0,C 180,E1 -15949.018,E2 -15949.018} C_VEL
LIN {X 0,Y 312.51,Z 354.159,A -85,B 0,C 180,E1 -15949.483,E2 -15949.483} C_VEL
LIN {X 0,Y 308.301,Z 329.321,A -85,B 0,C 180,E1 -15950.363,E2 -15950.363} C_VEL
LIN {X 0,Y 307.293,Z 324.05,A -85,B 0,C 180,E1 -15950.594,E2 -15950.594} C_VEL
LIN {X 0,Y 307.4,Z 322.158,A -85,B 0,C 180,E1 -15951.108,E2 -15951.108} C_VEL
LIN {X 0,Y 307.329,Z 317.285,A -85,B 0,C 180,E1 -15952.877,E2 -15952.877} C_VEL
LIN {X 0,Y 305.668,Z 308.061,A -85,B 0,C 180,E1 -15956.434,E2 -15956.434} C_VEL
LIN {X 0,Y 305.488,Z 307.272,A -85,B 0,C 180,E1 -15956.921,E2 -15956.921} C_VEL
LIN {X 0,Y 305.427,Z 307.248,A -85,B 0,C 180,E1 -15960.412,E2 -15960.412} C_VEL
LIN {X 0,Y 305.461,Z 307.242,A -85,B 0,C 180,E1 -15964.078,E2 -15964.078} C_VEL
LIN {X 0,Y 305.45,Z 307.247,A -85,B 0,C 180,E1 -15966.742,E2 -15966.742} C_VEL
LIN {X 0,Y 305.404,Z 307.247,A -85,B 0,C 180,E1 -15970.589,E2 -15970.589} C_VEL
LIN {X 0,Y 305.415,Z 307.251,A -85,B 0,C 180,E1 -15973.656,E2 -15973.656} C_VEL
LIN {X 0,Y 305.428,Z 307.248,A -85,B 0,C 180,E1 -15977.418,E2 -15977.418} C_VEL
LIN {X 0,Y 305.436,Z 307.236,A -85,B 0,C 180,E1 -15981.592,E2 -15981.592} C_VEL
LIN {X 0,Y 305.455,Z 307.247,A -85,B 0,C 180,E1 -15984.886,E2 -15984.886} C_VEL
LIN {X 0,Y 305.435,Z 307.25,A -85,B 0,C 180,E1 -15988.358,E2 -15988.358} C_VEL
LIN {X 0,Y 305.467,Z 307.245,A -85,B 0,C 180,E1 -15991.108,E2 -15991.108} C_VEL
LIN {X 0,Y 305.471,Z 307.245,A -85,B 0,C 180,E1 -15994.079,E2 -15994.079} C_VEL
LIN {X 0,Y 305.451,Z 307.243,A -85,B 0,C 180,E1 -15998.399,E2 -15998.399} C_VEL
LIN {X 0,Y 305.495,Z 307.241,A -85,B 0,C 180,E1 -16001.212,E2 -16001.212} C_VEL
LIN {X 0,Y 305.571,Z 307.226,A -85,B 0,C 180,E1 -16005.345,E2 -16005.345} C_VEL
LIN {X 0,Y 305.616,Z 307.225,A -85,B 0,C 180,E1 -16009.399,E2 -16009.399} C_VEL
LIN {X 0,Y 305.739,Z 307.214,A -85,B 0,C 180,E1 -16012.073,E2 -16012.073} C_VEL
LIN {X 0,Y 305.648,Z 307.214,A -85,B 0,C 180,E1 -16014.723,E2 -16014.723} C_VEL
LIN {X 0,Y 305.926,Z 307.188,A -85,B 0,C 180,E1 -16018.684,E2 -16018.684} C_VEL
LIN {X 0,Y 305.925,Z 307.188,A -85,B 0,C 180,E1 -16021.317,E2 -16021.317} C_VEL
LIN {X 0,Y 305.777,Z 307.203,A -85,B 0,C 180,E1 -16026.599,E2 -16026.599} C_VEL
LIN {X 0,Y 305.676,Z 307.219,A -85,B 0,C 180,E1 -16029.262,E2 -16029.262} C_VEL
LIN {X 0,Y 305.561,Z 307.229,A -85,B 0,C 180,E1 -16033.297,E2 -16033.297} C_VEL
LIN {X 0,Y 305.506,Z 307.241,A -85,B 0,C 180,E1 -16036.025,E2 -16036.025} C_VEL
LIN {X 0,Y 305.469,Z 307.242,A -85,B 0,C 180,E1 -16040.189,E2 -16040.189} C_VEL
LIN {X 0,Y 305.432,Z 307.248,A -85,B 0,C 180,E1 -16044.468,E2 -16044.468} C_VEL
LIN {X 0,Y 305.442,Z 307.251,A -85,B 0,C 180,E1 -16047.399,E2 -16047.399} C_VEL
LIN {X 0,Y 305.423,Z 307.246,A -85,B 0,C 180,E1 -16050.414,E2 -16050.414} C_VEL
LIN {X 0,Y 305.459,Z 307.245,A -85,B 0,C 180,E1 -16054.079,E2 -16054.079} C_VEL
LIN {X 0,Y 305.446,Z 307.244,A -85,B 0,C 180,E1 -16056.744,E2 -16056.744} C_VEL
LIN {X 0,Y 305.404,Z 307.241,A -85,B 0,C 180,E1 -16060.59,E2 -16060.59} C_VEL
LIN {X 0,Y 305.416,Z 307.252,A -85,B 0,C 180,E1 -16063.657,E2 -16063.657} C_VEL
LIN {X 0,Y 305.43,Z 307.242,A -85,B 0,C 180,E1 -16067.42,E2 -16067.42} C_VEL
LIN {X 0,Y 305.457,Z 307.246,A -85,B 0,C 180,E1 -16071.596,E2 -16071.596} C_VEL
LIN {X 0,Y 305.46,Z 307.242,A -85,B 0,C 180,E1 -16074.887,E2 -16074.887} C_VEL
LIN {X 0,Y 305.44,Z 307.251,A -85,B 0,C 180,E1 -16078.359,E2 -16078.359} C_VEL
LIN {X 0,Y 305.453,Z 307.234,A -85,B 0,C 180,E1 -16082.603,E2 -16082.603} C_VEL
LIN {X 0,Y 305.54,Z 307.577,A -85,B 0,C 180,E1 -16083.413,E2 -16083.413} C_VEL
LIN {X 0,Y 306.988,Z 315.014,A -85,B 0,C 180,E1 -16086.311,E2 -16086.311} C_VEL
LIN {X 0,Y 307.493,Z 319.114,A -85,B 0,C 180,E1 -16087.845,E2 -16087.845} C_VEL
LIN {X 0,Y 307.278,Z 323.694,A -85,B 0,C 180,E1 -16089.399,E2 -16089.399} C_VEL
LIN {X 0,Y 307.899,Z 327.243,A -85,B 0,C 180,E1 -16089.604,E2 -16089.604} C_VEL
LIN {X 0,Y 311.76,Z 348.969,A -85,B 0,C 180,E1 -16090.389,E2 -16090.389} C_VEL
LIN {X 0,Y 312.559,Z 354.766,A -85,B 0,C 180,E1 -16090.58,E2 -16090.58} C_VEL
LIN {X 0,Y 311.689,Z 400.012,A -85,B 0,C 180,E1 -16091.642,E2 -16091.642} C_VEL
LIN {X 0,Y 311.295,Z 408.971,A -85,B 0,C 180,E1 -16092,E2 -16092} C_VEL
LIN {X 0,Y 310.717,Z 418.501,A -85,B 0,C 180,E1 -16092.561,E2 -16092.561} C_VEL
LIN {X 0,Y 309.919,Z 428.51,A -85,B 0,C 180,E1 -16093.364,E2 -16093.364} C_VEL
LIN {X 0,Y 308.763,Z 438.892,A -85,B 0,C 180,E1 -16094.488,E2 -16094.488} C_VEL
LIN {X 0,Y 307.808,Z 447.035,A -85,B 0,C 180,E1 -16095.623,E2 -16095.623} C_VEL
LIN {X 0,Y 306.967,Z 453.753,A -85,B 0,C 180,E1 -16096.765,E2 -16096.765} C_VEL
LIN {X 0,Y 306.091,Z 460.117,A -85,B 0,C 180,E1 -16098.075,E2 -16098.075} C_VEL
LIN {X 0,Y 305.397,Z 465.407,A -85,B 0,C 180,E1 -16099.391,E2 -16099.391} C_VEL
LIN {X 0,Y 304.844,Z 469.825,A -85,B 0,C 180,E1 -16100.713,E2 -16100.713} C_VEL
LIN {X 0,Y 304.208,Z 475.021,A -85,B 0,C 180,E1 -16102.7,E2 -16102.7} C_VEL
LIN {X 0,Y 303.925,Z 477.47,A -85,B 0,C 180,E1 -16103.9,E2 -16103.9} C_VEL
LIN {X 0,Y 303.731,Z 480.61,A -85,B 0,C 180,E1 -16106.02,E2 -16106.02} C_VEL
LIN {X 0,Y 303.626,Z 481.887,A -85,B 0,C 180,E1 -16107.347,E2 -16107.347} C_VEL
LIN {X 0,Y 303.538,Z 482.692,A -85,B 0,C 180,E1 -16108.673,E2 -16108.673} C_VEL
LIN {X 0,Y 303.511,Z 482.998,A -85,B 0,C 180,E1 -16110,E2 -16110} C_VEL
LIN {X 0,Y 303.534,Z 482.719,A -85,B 0,C 180,E1 -16111.327,E2 -16111.327} C_VEL
LIN {X 0,Y 303.614,Z 481.969,A -85,B 0,C 180,E1 -16112.653,E2 -16112.653} C_VEL
LIN {X 0,Y 303.707,Z 480.748,A -85,B 0,C 180,E1 -16113.981,E2 -16113.981} C_VEL
LIN {X 0,Y 303.832,Z 479.035,A -85,B 0,C 180,E1 -16115.309,E2 -16115.309} C_VEL
LIN {X 0,Y 304.202,Z 475.278,A -85,B 0,C 180,E1 -16117.3,E2 -16117.3} C_VEL
LIN {X 0,Y 304.793,Z 470.15,A -85,B 0,C 180,E1 -16119.288,E2 -16119.288} C_VEL
LIN {X 0,Y 305.54,Z 464.635,A -85,B 0,C 180,E1 -16120.939,E2 -16120.939} C_VEL
LIN {X 0,Y 306.473,Z 457.708,A -85,B 0,C 180,E1 -16122.583,E2 -16122.583} C_VEL
LIN {X 0,Y 307.473,Z 449.755,A -85,B 0,C 180,E1 -16124.055,E2 -16124.055} C_VEL
LIN {X 0,Y 308.425,Z 442.173,A -85,B 0,C 180,E1 -16125.191,E2 -16125.191} C_VEL
LIN {X 0,Y 309.359,Z 434.227,A -85,B 0,C 180,E1 -16126.158,E2 -16126.158} C_VEL
LIN {X 0,Y 310.146,Z 426.018,A -85,B 0,C 180,E1 -16126.962,E2 -16126.962} C_VEL
LIN {X 0,Y 310.853,Z 417.698,A -85,B 0,C 180,E1 -16127.601,E2 -16127.601} C_VEL
LIN {X 0,Y 311.328,Z 408.699,A -85,B 0,C 180,E1 -16128.125,E2 -16128.125} C_VEL
LIN {X 0,Y 311.725,Z 399.302,A -85,B 0,C 180,E1 -16128.493,E2 -16128.493} C_VEL
LIN {X 0,Y 312.435,Z 353.287,A -85,B 0,C 180,E1 -16129.578,E2 -16129.578} C_VEL
LIN {X 0,Y 308.588,Z 330.756,A -85,B 0,C 180,E1 -16130.379,E2 -16130.379} C_VEL
LIN {X 0,Y 307.321,Z 324.194,A -85,B 0,C 180,E1 -16130.657,E2 -16130.657} C_VEL
LIN {X 0,Y 307.289,Z 323.418,A -85,B 0,C 180,E1 -16130.775,E2 -16130.775} C_VEL
LIN {X 0,Y 307.496,Z 319.434,A -85,B 0,C 180,E1 -16132.155,E2 -16132.155} C_VEL
LIN {X 0,Y 306.741,Z 313.577,A -85,B 0,C 180,E1 -16134.356,E2 -16134.356} C_VEL
LIN {X 0,Y 305.531,Z 307.331,A -85,B 0,C 180,E1 -16136.84,E2 -16136.84} C_VEL
LIN {X 0,Y 305.428,Z 307.248,A -85,B 0,C 180,E1 -16140.412,E2 -16140.412} C_VEL
LIN {X 0,Y 305.463,Z 307.242,A -85,B 0,C 180,E1 -16144.078,E2 -16144.078} C_VEL
LIN {X 0,Y 305.451,Z 307.246,A -85,B 0,C 180,E1 -16146.742,E2 -16146.742} C_VEL
LIN {X 0,Y 305.405,Z 307.247,A -85,B 0,C 180,E1 -16150.589,E2 -16150.589} C_VEL
LIN {X 0,Y 305.416,Z 307.251,A -85,B 0,C 180,E1 -16153.655,E2 -16153.655} C_VEL
LIN {X 0,Y 305.43,Z 307.249,A -85,B 0,C 180,E1 -16157.418,E2 -16157.418} C_VEL
LIN {X 0,Y 305.439,Z 307.235,A -85,B 0,C 180,E1 -16161.592,E2 -16161.592} C_VEL
LIN {X 0,Y 305.412,Z 307.239,A -85,B 0,C 180,E1 -16162.538,E2 -16162.538} C_VEL
LIN {X 0,Y 304.764,Z 307.328,A -85,B 0,C 180,E1 -16163.638,E2 -16163.638} C_VEL
LIN {X 0,Y 301.923,Z 307.687,A -85,B 0,C 180,E1 -16165.429,E2 -16165.429} C_VEL
LIN {X 0,Y 299.5,Z 307.993,A -85,B 0,C 180,E1 -16166.881,E2 -16166.881} C_VEL
LIN {X 0,Y 298.456,Z 308.118,A -85,B 0,C 180,E1 -16168.006,E2 -16168.006} C_VEL
LIN {X 0,Y 298.37,Z 308.128,A -85,B 0,C 180,E1 -16168.388,E2 -16168.388} C_VEL
LIN {X 0,Y 298.403,Z 308.122,A -85,B 0,C 180,E1 -16171.898,E2 -16171.898} C_VEL
LIN {X 0,Y 298.406,Z 308.126,A -85,B 0,C 180,E1 -16174.917,E2 -16174.917} C_VEL
LIN {X 0,Y 298.384,Z 308.12,A -85,B 0,C 180,E1 -16177.861,E2 -16177.861} C_VEL
LIN {X 0,Y 298.446,Z 308.122,A -85,B 0,C 180,E1 -16180.75,E2 -16180.75} C_VEL
LIN {X 0,Y 298.503,Z 308.107,A -85,B 0,C 180,E1 -16184.99,E2 -16184.99} C_VEL
LIN {X 0,Y 298.575,Z 308.102,A -85,B 0,C 180,E1 -16189.146,E2 -16189.146} C_VEL
LIN {X 0,Y 298.69,Z 308.091,A -85,B 0,C 180,E1 -16191.884,E2 -16191.884} C_VEL
LIN {X 0,Y 298.618,Z 308.09,A -85,B 0,C 180,E1 -16194.598,E2 -16194.598} C_VEL
LIN {X 0,Y 298.894,Z 308.064,A -85,B 0,C 180,E1 -16198.653,E2 -16198.653} C_VEL
LIN {X 0,Y 298.893,Z 308.064,A -85,B 0,C 180,E1 -16201.347,E2 -16201.347} C_VEL
LIN {X 0,Y 298.725,Z 308.081,A -85,B 0,C 180,E1 -16206.755,E2 -16206.755} C_VEL
LIN {X 0,Y 298.609,Z 308.101,A -85,B 0,C 180,E1 -16209.483,E2 -16209.483} C_VEL
LIN {X 0,Y 298.514,Z 308.106,A -85,B 0,C 180,E1 -16213.617,E2 -16213.617} C_VEL
LIN {X 0,Y 298.446,Z 308.118,A -85,B 0,C 180,E1 -16216.414,E2 -16216.414} C_VEL
LIN {X 0,Y 298.425,Z 308.123,A -85,B 0,C 180,E1 -16219.611,E2 -16219.611} C_VEL
LIN {X 0,Y 298.375,Z 308.128,A -85,B 0,C 180,E1 -16223.604,E2 -16223.604} C_VEL
LIN {X 0,Y 298.395,Z 308.126,A -85,B 0,C 180,E1 -16226.583,E2 -16226.583} C_VEL
LIN {X 0,Y 298.386,Z 308.124,A -85,B 0,C 180,E1 -16229.645,E2 -16229.645} C_VEL
LIN {X 0,Y 298.387,Z 308.129,A -85,B 0,C 180,E1 -16232.801,E2 -16232.801} C_VEL
LIN {X 0,Y 298.42,Z 308.116,A -85,B 0,C 180,E1 -16236.802,E2 -16236.802} C_VEL
LIN {X 0,Y 298.368,Z 308.112,A -85,B 0,C 180,E1 -16239.492,E2 -16239.492} C_VEL
LIN {X 0,Y 298.364,Z 308.133,A -85,B 0,C 180,E1 -16243.098,E2 -16243.098} C_VEL
LIN {X 0,Y 298.364,Z 308.124,A -85,B 0,C 180,E1 -16246.915,E2 -16246.915} C_VEL
LIN {X 0,Y 298.38,Z 308.13,A -85,B 0,C 180,E1 -16251.012,E2 -16251.012} C_VEL
LIN {X 0,Y 298.401,Z 308.124,A -85,B 0,C 180,E1 -16253.929,E2 -16253.929} C_VEL
LIN {X 0,Y 298.39,Z 308.129,A -85,B 0,C 180,E1 -16257.2,E2 -16257.2} C_VEL
LIN {X 0,Y 298.399,Z 308.131,A -85,B 0,C 180,E1 -16260.626,E2 -16260.626} C_VEL
LIN {X 0,Y 298.447,Z 308.225,A -85,B 0,C 180,E1 -16262.875,E2 -16262.875} C_VEL
LIN {X 0,Y 300.22,Z 317.36,A -85,B 0,C 180,E1 -16266.55,E2 -16266.55} C_VEL
LIN {X 0,Y 300.49,Z 322.238,A -85,B 0,C 180,E1 -16268.385,E2 -16268.385} C_VEL
LIN {X 0,Y 300.413,Z 323.841,A -85,B 0,C 180,E1 -16268.861,E2 -16268.861} C_VEL
LIN {X 0,Y 302.21,Z 333.168,A -85,B 0,C 180,E1 -16269.277,E2 -16269.277} C_VEL
LIN {X 0,Y 305.696,Z 353.74,A -85,B 0,C 180,E1 -16270.029,E2 -16270.029} C_VEL
LIN {X 0,Y 305.723,Z 363.717,A -85,B 0,C 180,E1 -16270.275,E2 -16270.275} C_VEL
LIN {X 0,Y 304.995,Z 400.828,A -85,B 0,C 180,E1 -16271.18,E2 -16271.18} C_VEL
LIN {X 0,Y 304.433,Z 411.981,A -85,B 0,C 180,E1 -16271.667,E2 -16271.667} C_VEL
LIN {X 0,Y 303.607,Z 423.654,A -85,B 0,C 180,E1 -16272.487,E2 -16272.487} C_VEL
LIN {X 0,Y 302.692,Z 432.332,A -85,B 0,C 180,E1 -16273.302,E2 -16273.302} C_VEL
LIN {X 0,Y 301.77,Z 440.621,A -85,B 0,C 180,E1 -16274.292,E2 -16274.292} C_VEL
LIN {X 0,Y 300.747,Z 448.465,A -85,B 0,C 180,E1 -16275.451,E2 -16275.451} C_VEL
LIN {X 0,Y 299.807,Z 455.799,A -85,B 0,C 180,E1 -16276.788,E2 -16276.788} C_VEL
LIN {X 0,Y 298.721,Z 463.237,A -85,B 0,C 180,E1 -16278.465,E2 -16278.465} C_VEL
LIN {X 0,Y 297.791,Z 470.023,A -85,B 0,C 180,E1 -16280.491,E2 -16280.491} C_VEL
LIN {X 0,Y 297.158,Z 475.176,A -85,B 0,C 180,E1 -16282.526,E2 -16282.526} C_VEL
LIN {X 0,Y 296.769,Z 478.958,A -85,B 0,C 180,E1 -16284.565,E2 -16284.565} C_VEL
LIN {X 0,Y 296.647,Z 480.694,A -85,B 0,C 180,E1 -16285.924,E2 -16285.924} C_VEL
LIN {X 0,Y 296.553,Z 481.936,A -85,B 0,C 180,E1 -16287.283,E2 -16287.283} C_VEL
LIN {X 0,Y 296.459,Z 482.708,A -85,B 0,C 180,E1 -16288.642,E2 -16288.642} C_VEL
LIN {X 0,Y 296.429,Z 483,A -85,B 0,C 180,E1 -16290,E2 -16290} C_VEL
LIN {X 0,Y 296.459,Z 482.702,A -85,B 0,C 180,E1 -16291.358,E2 -16291.358} C_VEL
LIN {X 0,Y 296.553,Z 481.919,A -85,B 0,C 180,E1 -16292.717,E2 -16292.717} C_VEL
LIN {X 0,Y 296.646,Z 480.665,A -85,B 0,C 180,E1 -16294.076,E2 -16294.076} C_VEL
LIN {X 0,Y 296.833,Z 477.864,A -85,B 0,C 180,E1 -16296.058,E2 -16296.058} C_VEL
LIN {X 0,Y 297.159,Z 475.123,A -85,B 0,C 180,E1 -16297.474,E2 -16297.474} C_VEL
LIN {X 0,Y 297.789,Z 469.952,A -85,B 0,C 180,E1 -16299.509,E2 -16299.509} C_VEL
LIN {X 0,Y 298.716,Z 463.134,A -85,B 0,C 180,E1 -16301.536,E2 -16301.536} C_VEL
LIN {X 0,Y 299.805,Z 455.679,A -85,B 0,C 180,E1 -16303.212,E2 -16303.212} C_VEL
LIN {X 0,Y 300.767,Z 448.325,A -85,B 0,C 180,E1 -16304.548,E2 -16304.548} C_VEL
LIN {X 0,Y 301.771,Z 440.446,A -85,B 0,C 180,E1 -16305.708,E2 -16305.708} C_VEL
LIN {X 0,Y 302.743,Z 432.116,A -85,B 0,C 180,E1 -16306.695,E2 -16306.695} C_VEL
LIN {X 0,Y 303.713,Z 421.464,A -85,B 0,C 180,E1 -16307.681,E2 -16307.681} C_VEL
LIN {X 0,Y 304.456,Z 410.673,A -85,B 0,C 180,E1 -16308.375,E2 -16308.375} C_VEL
LIN {X 0,Y 304.942,Z 401.369,A -85,B 0,C 180,E1 -16308.78,E2 -16308.78} C_VEL
LIN {X 0,Y 305.505,Z 373.684,A -85,B 0,C 180,E1 -16309.47,E2 -16309.47} C_VEL
LIN {X 0,Y 305.716,Z 354.318,A -85,B 0,C 180,E1 -16309.93,E2 -16309.93} C_VEL
LIN {X 0,Y 301.667,Z 330.396,A -85,B 0,C 180,E1 -16310.804,E2 -16310.804} C_VEL
LIN {X 0,Y 300.417,Z 323.863,A -85,B 0,C 180,E1 -16311.109,E2 -16311.109} C_VEL
LIN {X 0,Y 300.518,Z 321.188,A -85,B 0,C 180,E1 -16311.973,E2 -16311.973} C_VEL
LIN {X 0,Y 299.78,Z 314.931,A -85,B 0,C 180,E1 -16314.372,E2 -16314.372} C_VEL
LIN {X 0,Y 298.449,Z 308.204,A -85,B 0,C 180,E1 -16317.125,E2 -16317.125} C_VEL
LIN {X 0,Y 298.374,Z 308.126,A -85,B 0,C 180,E1 -16321.21,E2 -16321.21} C_VEL
LIN {X 0,Y 298.425,Z 308.118,A -85,B 0,C 180,E1 -16324.487,E2 -16324.487} C_VEL
LIN {X 0,Y 298.394,Z 308.128,A -85,B 0,C 180,E1 -16327.76,E2 -16327.76} C_VEL
LIN {X 0,Y 298.341,Z 308.122,A -85,B 0,C 180,E1 -16331.268,E2 -16331.268} C_VEL
LIN {X 0,Y 298.35,Z 308.134,A -85,B 0,C 180,E1 -16335.034,E2 -16335.034} C_VEL
LIN {X 0,Y 298.342,Z 308.124,A -85,B 0,C 180,E1 -16338.921,E2 -16338.921} C_VEL
LIN {X 0,Y 298.381,Z 308.113,A -85,B 0,C 180,E1 -16342.237,E2 -16342.237} C_VEL
LIN {X 0,Y 298.402,Z 308.125,A -85,B 0,C 180,E1 -16345.58,E2 -16345.58} C_VEL
LIN {X 0,Y 298.37,Z 308.129,A -85,B 0,C 180,E1 -16348.788,E2 -16348.788} C_VEL
LIN {X 0,Y 298.402,Z 308.123,A -85,B 0,C 180,E1 -16351.898,E2 -16351.898} C_VEL
LIN {X 0,Y 298.406,Z 308.126,A -85,B 0,C 180,E1 -16354.917,E2 -16354.917} C_VEL
LIN {X 0,Y 298.383,Z 308.12,A -85,B 0,C 180,E1 -16357.861,E2 -16357.861} C_VEL
LIN {X 0,Y 298.446,Z 308.122,A -85,B 0,C 180,E1 -16360.751,E2 -16360.751} C_VEL
LIN {X 0,Y 298.503,Z 308.107,A -85,B 0,C 180,E1 -16364.99,E2 -16364.99} C_VEL
LIN {X 0,Y 298.574,Z 308.102,A -85,B 0,C 180,E1 -16369.146,E2 -16369.146} C_VEL
LIN {X 0,Y 298.69,Z 308.091,A -85,B 0,C 180,E1 -16371.884,E2 -16371.884} C_VEL
LIN {X 0,Y 298.618,Z 308.089,A -85,B 0,C 180,E1 -16374.598,E2 -16374.598} C_VEL
LIN {X 0,Y 298.894,Z 308.064,A -85,B 0,C 180,E1 -16378.653,E2 -16378.653} C_VEL
LIN {X 0,Y 298.893,Z 308.064,A -85,B 0,C 180,E1 -16381.347,E2 -16381.347} C_VEL
LIN {X 0,Y 298.725,Z 308.081,A -85,B 0,C 180,E1 -16386.756,E2 -16386.756} C_VEL
LIN {X 0,Y 298.609,Z 308.101,A -85,B 0,C 180,E1 -16389.483,E2 -16389.483} C_VEL
LIN {X 0,Y 298.514,Z 308.106,A -85,B 0,C 180,E1 -16393.617,E2 -16393.617} C_VEL
LIN {X 0,Y 298.446,Z 308.118,A -85,B 0,C 180,E1 -16396.415,E2 -16396.415} C_VEL
LIN {X 0,Y 298.425,Z 308.124,A -85,B 0,C 180,E1 -16399.612,E2 -16399.612} C_VEL
LIN {X 0,Y 298.375,Z 308.128,A -85,B 0,C 180,E1 -16403.605,E2 -16403.605} C_VEL
LIN {X 0,Y 298.396,Z 308.126,A -85,B 0,C 180,E1 -16406.584,E2 -16406.584} C_VEL
LIN {X 0,Y 298.386,Z 308.123,A -85,B 0,C 180,E1 -16409.645,E2 -16409.645} C_VEL
LIN {X 0,Y 298.387,Z 308.128,A -85,B 0,C 180,E1 -16412.801,E2 -16412.801} C_VEL
LIN {X 0,Y 298.398,Z 308.12,A -85,B 0,C 180,E1 -16416.073,E2 -16416.073} C_VEL
LIN {X 0,Y 298.369,Z 308.112,A -85,B 0,C 180,E1 -16419.493,E2 -16419.493} C_VEL
LIN {X 0,Y 298.365,Z 308.132,A -85,B 0,C 180,E1 -16423.098,E2 -16423.098} C_VEL
LIN {X 0,Y 298.366,Z 308.125,A -85,B 0,C 180,E1 -16426.915,E2 -16426.915} C_VEL
LIN {X 0,Y 298.382,Z 308.129,A -85,B 0,C 180,E1 -16431.012,E2 -16431.012} C_VEL
LIN {X 0,Y 298.403,Z 308.124,A -85,B 0,C 180,E1 -16433.929,E2 -16433.929} C_VEL
LIN {X 0,Y 298.391,Z 308.129,A -85,B 0,C 180,E1 -16437.2,E2 -16437.2} C_VEL
LIN {X 0,Y 298.362,Z 308.135,A -85,B 0,C 180,E1 -16440.639,E2 -16440.639} C_VEL
LIN {X 0,Y 298.429,Z 308.281,A -85,B 0,C 180,E1 -16442.977,E2 -16442.977} C_VEL
LIN {X 0,Y 299.945,Z 315.861,A -85,B 0,C 180,E1 -16446.037,E2 -16446.037} C_VEL
LIN {X 0,Y 300.517,Z 321.067,A -85,B 0,C 180,E1 -16448.027,E2 -16448.027} C_VEL
LIN {X 0,Y 300.408,Z 323.947,A -85,B 0,C 180,E1 -16448.946,E2 -16448.946} C_VEL
LIN {X 0,Y 304.047,Z 343.54,A -85,B 0,C 180,E1 -16449.736,E2 -16449.736} C_VEL
LIN {X 0,Y 305.832,Z 355.134,A -85,B 0,C 180,E1 -16450.143,E2 -16450.143} C_VEL
LIN {X 0,Y 304.961,Z 400.03,A -85,B 0,C 180,E1 -16451.222,E2 -16451.222} C_VEL
LIN {X 0,Y 304.559,Z 408.982,A -85,B 0,C 180,E1 -16451.588,E2 -16451.588} C_VEL
LIN {X 0,Y 303.975,Z 418.509,A -85,B 0,C 180,E1 -16452.161,E2 -16452.161} C_VEL
LIN {X 0,Y 303.134,Z 428.517,A -85,B 0,C 180,E1 -16452.98,E2 -16452.98} C_VEL
LIN {X 0,Y 301.945,Z 438.896,A -85,B 0,C 180,E1 -16454.128,E2 -16454.128} C_VEL
LIN {X 0,Y 300.952,Z 447.038,A -85,B 0,C 180,E1 -16455.288,E2 -16455.288} C_VEL
LIN {X 0,Y 300.045,Z 453.756,A -85,B 0,C 180,E1 -16456.454,E2 -16456.454} C_VEL
LIN {X 0,Y 299.145,Z 460.119,A -85,B 0,C 180,E1 -16457.793,E2 -16457.793} C_VEL
LIN {X 0,Y 298.423,Z 465.409,A -85,B 0,C 180,E1 -16459.141,E2 -16459.141} C_VEL
LIN {X 0,Y 297.84,Z 469.827,A -85,B 0,C 180,E1 -16460.493,E2 -16460.493} C_VEL
LIN {X 0,Y 297.166,Z 475.023,A -85,B 0,C 180,E1 -16462.526,E2 -16462.526} C_VEL
LIN {X 0,Y 296.84,Z 477.771,A -85,B 0,C 180,E1 -16463.932,E2 -16463.932} C_VEL
LIN {X 0,Y 296.652,Z 480.611,A -85,B 0,C 180,E1 -16465.924,E2 -16465.924} C_VEL
LIN {X 0,Y 296.555,Z 481.887,A -85,B 0,C 180,E1 -16467.283,E2 -16467.283} C_VEL
LIN {X 0,Y 296.46,Z 482.692,A -85,B 0,C 180,E1 -16468.642,E2 -16468.642} C_VEL
LIN {X 0,Y 296.43,Z 482.998,A -85,B 0,C 180,E1 -16470,E2 -16470} C_VEL
LIN {X 0,Y 296.456,Z 482.719,A -85,B 0,C 180,E1 -16471.358,E2 -16471.358} C_VEL
LIN {X 0,Y 296.543,Z 481.968,A -85,B 0,C 180,E1 -16472.717,E2 -16472.717} C_VEL
LIN {X 0,Y 296.629,Z 480.748,A -85,B 0,C 180,E1 -16474.076,E2 -16474.076} C_VEL
LIN {X 0,Y 296.874,Z 477.86,A -85,B 0,C 180,E1 -16476.129,E2 -16476.129} C_VEL
LIN {X 0,Y 297.16,Z 475.276,A -85,B 0,C 180,E1 -16477.474,E2 -16477.474} C_VEL
LIN {X 0,Y 297.768,Z 470.148,A -85,B 0,C 180,E1 -16479.51,E2 -16479.51} C_VEL
LIN {X 0,Y 298.542,Z 464.633,A -85,B 0,C 180,E1 -16481.199,E2 -16481.199} C_VEL
LIN {X 0,Y 299.55,Z 457.705,A -85,B 0,C 180,E1 -16482.878,E2 -16482.878} C_VEL
LIN {X 0,Y 300.579,Z 449.751,A -85,B 0,C 180,E1 -16484.384,E2 -16484.384} C_VEL
LIN {X 0,Y 301.596,Z 442.169,A -85,B 0,C 180,E1 -16485.544,E2 -16485.544} C_VEL
LIN {X 0,Y 302.552,Z 434.221,A -85,B 0,C 180,E1 -16486.532,E2 -16486.532} C_VEL
LIN {X 0,Y 303.359,Z 426.012,A -85,B 0,C 180,E1 -16487.354,E2 -16487.354} C_VEL
LIN {X 0,Y 304.099,Z 417.689,A -85,B 0,C 180,E1 -16488.005,E2 -16488.005} C_VEL
LIN {X 0,Y 304.582,Z 408.687,A -85,B 0,C 180,E1 -16488.541,E2 -16488.541} C_VEL
LIN {X 0,Y 305.026,Z 398.89,A -85,B 0,C 180,E1 -16488.928,E2 -16488.928} C_VEL
LIN {X 0,Y 305.76,Z 354.212,A -85,B 0,C 180,E1 -16490,E2 -16490} C_VEL
LIN {X 0,Y 301.748,Z 330.727,A -85,B 0,C 180,E1 -16490.862,E2 -16490.862} C_VEL
LIN {X 0,Y 300.442,Z 323.816,A -85,B 0,C 180,E1 -16491.186,E2 -16491.186} C_VEL
LIN {X 0,Y 300.517,Z 321.385,A -85,B 0,C 180,E1 -16491.973,E2 -16491.973} C_VEL
LIN {X 0,Y 299.82,Z 315.103,A -85,B 0,C 180,E1 -16494.378,E2 -16494.378} C_VEL
LIN {X 0,Y 298.467,Z 308.19,A -85,B 0,C 180,E1 -16497.228,E2 -16497.228} C_VEL
LIN {X 0,Y 298.375,Z 308.126,A -85,B 0,C 180,E1 -16501.21,E2 -16501.21} C_VEL
LIN {X 0,Y 298.427,Z 308.118,A -85,B 0,C 180,E1 -16504.487,E2 -16504.487} C_VEL
LIN {X 0,Y 298.395,Z 308.128,A -85,B 0,C 180,E1 -16507.76,E2 -16507.76} C_VEL
LIN {X 0,Y 298.343,Z 308.121,A -85,B 0,C 180,E1 -16511.267,E2 -16511.267} C_VEL
LIN {X 0,Y 298.351,Z 308.134,A -85,B 0,C 180,E1 -16515.034,E2 -16515.034} C_VEL
LIN {X 0,Y 298.343,Z 308.125,A -85,B 0,C 180,E1 -16518.92,E2 -16518.92} C_VEL
LIN {X 0,Y 298.421,Z 308.115,A -85,B 0,C 180,E1 -16523.197,E2 -16523.197} C_VEL
LIN {X 0,Y 298.387,Z 308.129,A -85,B 0,C 180,E1 -16527.199,E2 -16527.199} C_VEL
LIN {X 0,Y 298.37,Z 308.128,A -85,B 0,C 180,E1 -16528.388,E2 -16528.388} C_VEL
LIN {X 0,Y 297.711,Z 308.213,A -85,B 0,C 180,E1 -16529.513,E2 -16529.513} C_VEL
LIN {X 0,Y 294.901,Z 308.57,A -85,B 0,C 180,E1 -16531.348,E2 -16531.348} C_VEL
LIN {X 0,Y 292.496,Z 308.87,A -85,B 0,C 180,E1 -16532.836,E2 -16532.836} C_VEL
LIN {X 0,Y 291.432,Z 308.997,A -85,B 0,C 180,E1 -16533.987,E2 -16533.987} C_VEL
LIN {X 0,Y 291.328,Z 309.007,A -85,B 0,C 180,E1 -16534.378,E2 -16534.378} C_VEL
LIN {X 0,Y 291.343,Z 308.996,A -85,B 0,C 180,E1 -16537.296,E2 -16537.296} C_VEL
LIN {X 0,Y 291.378,Z 308.999,A -85,B 0,C 180,E1 -16540.264,E2 -16540.264} C_VEL
LIN {X 0,Y 291.468,Z 308.984,A -85,B 0,C 180,E1 -16544.682,E2 -16544.682} C_VEL
LIN {X 0,Y 291.52,Z 308.982,A -85,B 0,C 180,E1 -16548.88,E2 -16548.88} C_VEL
LIN {X 0,Y 291.644,Z 308.967,A -85,B 0,C 180,E1 -16551.686,E2 -16551.686} C_VEL
LIN {X 0,Y 291.588,Z 308.965,A -85,B 0,C 180,E1 -16554.467,E2 -16554.467} C_VEL
LIN {X 0,Y 291.862,Z 308.94,A -85,B 0,C 180,E1 -16558.62,E2 -16558.62} C_VEL
LIN {X 0,Y 291.86,Z 308.94,A -85,B 0,C 180,E1 -16561.38,E2 -16561.38} C_VEL
LIN {X 0,Y 291.676,Z 308.959,A -85,B 0,C 180,E1 -16566.919,E2 -16566.919} C_VEL
LIN {X 0,Y 291.555,Z 308.982,A -85,B 0,C 180,E1 -16569.714,E2 -16569.714} C_VEL
LIN {X 0,Y 291.473,Z 308.982,A -85,B 0,C 180,E1 -16573.953,E2 -16573.953} C_VEL
LIN {X 0,Y 291.397,Z 308.996,A -85,B 0,C 180,E1 -16576.823,E2 -16576.823} C_VEL
LIN {X 0,Y 291.385,Z 308.998,A -85,B 0,C 180,E1 -16579.842,E2 -16579.842} C_VEL
LIN {X 0,Y 291.319,Z 309.006,A -85,B 0,C 180,E1 -16584.212,E2 -16584.212} C_VEL
LIN {X 0,Y 291.343,Z 309.007,A -85,B 0,C 180,E1 -16587.279,E2 -16587.279} C_VEL
LIN {X 0,Y 291.312,Z 309.003,A -85,B 0,C 180,E1 -16590.44,E2 -16590.44} C_VEL
LIN {X 0,Y 291.338,Z 309.006,A -85,B 0,C 180,E1 -16593.699,E2 -16593.699} C_VEL
LIN {X 0,Y 291.342,Z 308.99,A -85,B 0,C 180,E1 -16597.247,E2 -16597.247} C_VEL
LIN {X 0,Y 291.294,Z 308.997,A -85,B 0,C 180,E1 -16600.649,E2 -16600.649} C_VEL
LIN {X 0,Y 291.277,Z 309.014,A -85,B 0,C 180,E1 -16604.404,E2 -16604.404} C_VEL
LIN {X 0,Y 291.289,Z 308.998,A -85,B 0,C 180,E1 -16608.412,E2 -16608.412} C_VEL
LIN {X 0,Y 291.33,Z 309.008,A -85,B 0,C 180,E1 -16611.156,E2 -16611.156} C_VEL
LIN {X 0,Y 291.352,Z 308.998,A -85,B 0,C 180,E1 -16614.626,E2 -16614.626} C_VEL
LIN {X 0,Y 291.363,Z 309.004,A -85,B 0,C 180,E1 -16617.95,E2 -16617.95} C_VEL
LIN {X 0,Y 291.434,Z 309.082,A -85,B 0,C 180,E1 -16622.487,E2 -16622.487} C_VEL
LIN {X 0,Y 293.01,Z 317.362,A -85,B 0,C 180,E1 -16625.937,E2 -16625.937} C_VEL
LIN {X 0,Y 293.536,Z 322.24,A -85,B 0,C 180,E1 -16627.846,E2 -16627.846} C_VEL
LIN {X 0,Y 293.558,Z 323.974,A -85,B 0,C 180,E1 -16628.356,E2 -16628.356} C_VEL
LIN {X 0,Y 296.926,Z 341.394,A -85,B 0,C 180,E1 -16629.099,E2 -16629.099} C_VEL
LIN {X 0,Y 299.192,Z 355.842,A -85,B 0,C 180,E1 -16629.628,E2 -16629.628} C_VEL
LIN {X 0,Y 298.351,Z 400.049,A -85,B 0,C 180,E1 -16630.717,E2 -16630.717} C_VEL
LIN {X 0,Y 297.84,Z 409.501,A -85,B 0,C 180,E1 -16631.113,E2 -16631.113} C_VEL
LIN {X 0,Y 297.142,Z 419.49,A -85,B 0,C 180,E1 -16631.737,E2 -16631.737} C_VEL
LIN {X 0,Y 296.109,Z 430.836,A -85,B 0,C 180,E1 -16632.742,E2 -16632.742} C_VEL
LIN {X 0,Y 295.124,Z 439.395,A -85,B 0,C 180,E1 -16633.751,E2 -16633.751} C_VEL
LIN {X 0,Y 294.006,Z 447.448,A -85,B 0,C 180,E1 -16634.933,E2 -16634.933} C_VEL
LIN {X 0,Y 293.1,Z 454.098,A -85,B 0,C 180,E1 -16636.127,E2 -16636.127} C_VEL
LIN {X 0,Y 292.191,Z 460.41,A -85,B 0,C 180,E1 -16637.498,E2 -16637.498} C_VEL
LIN {X 0,Y 291.411,Z 465.653,A -85,B 0,C 180,E1 -16638.876,E2 -16638.876} C_VEL
LIN {X 0,Y 290.79,Z 470.024,A -85,B 0,C 180,E1 -16640.26,E2 -16640.26} C_VEL
LIN {X 0,Y 290.11,Z 475.178,A -85,B 0,C 180,E1 -16642.343,E2 -16642.343} C_VEL
LIN {X 0,Y 289.692,Z 478.959,A -85,B 0,C 180,E1 -16644.431,E2 -16644.431} C_VEL
LIN {X 0,Y 289.552,Z 480.695,A -85,B 0,C 180,E1 -16645.824,E2 -16645.824} C_VEL
LIN {X 0,Y 289.463,Z 481.937,A -85,B 0,C 180,E1 -16647.217,E2 -16647.217} C_VEL
LIN {X 0,Y 289.384,Z 482.708,A -85,B 0,C 180,E1 -16648.608,E2 -16648.608} C_VEL
LIN {X 0,Y 289.351,Z 483,A -85,B 0,C 180,E1 -16650,E2 -16650} C_VEL
LIN {X 0,Y 289.384,Z 482.702,A -85,B 0,C 180,E1 -16651.392,E2 -16651.392} C_VEL
LIN {X 0,Y 289.462,Z 481.919,A -85,B 0,C 180,E1 -16652.783,E2 -16652.783} C_VEL
LIN {X 0,Y 289.55,Z 480.664,A -85,B 0,C 180,E1 -16654.176,E2 -16654.176} C_VEL
LIN {X 0,Y 289.746,Z 478.167,A -85,B 0,C 180,E1 -16656.022,E2 -16656.022} C_VEL
LIN {X 0,Y 290.111,Z 475.121,A -85,B 0,C 180,E1 -16657.657,E2 -16657.657} C_VEL
LIN {X 0,Y 290.787,Z 469.951,A -85,B 0,C 180,E1 -16659.74,E2 -16659.74} C_VEL
LIN {X 0,Y 291.766,Z 463.132,A -85,B 0,C 180,E1 -16661.814,E2 -16661.814} C_VEL
LIN {X 0,Y 292.899,Z 455.677,A -85,B 0,C 180,E1 -16663.529,E2 -16663.529} C_VEL
LIN {X 0,Y 293.889,Z 448.322,A -85,B 0,C 180,E1 -16664.896,E2 -16664.896} C_VEL
LIN {X 0,Y 294.953,Z 440.442,A -85,B 0,C 180,E1 -16666.081,E2 -16666.081} C_VEL
LIN {X 0,Y 295.943,Z 432.111,A -85,B 0,C 180,E1 -16667.09,E2 -16667.09} C_VEL
LIN {X 0,Y 296.963,Z 421.458,A -85,B 0,C 180,E1 -16668.096,E2 -16668.096} C_VEL
LIN {X 0,Y 297.743,Z 410.663,A -85,B 0,C 180,E1 -16668.804,E2 -16668.804} C_VEL
LIN {X 0,Y 298.236,Z 401.354,A -85,B 0,C 180,E1 -16669.218,E2 -16669.218} C_VEL
LIN {X 0,Y 298.826,Z 373.677,A -85,B 0,C 180,E1 -16669.923,E2 -16669.923} C_VEL
LIN {X 0,Y 299.029,Z 354.985,A -85,B 0,C 180,E1 -16670.378,E2 -16670.378} C_VEL
LIN {X 0,Y 295.056,Z 331.542,A -85,B 0,C 180,E1 -16671.263,E2 -16671.263} C_VEL
LIN {X 0,Y 293.534,Z 323.889,A -85,B 0,C 180,E1 -16671.624,E2 -16671.624} C_VEL
LIN {X 0,Y 293.493,Z 321.187,A -85,B 0,C 180,E1 -16672.528,E2 -16672.528} C_VEL
LIN {X 0,Y 292.63,Z 315.332,A -85,B 0,C 180,E1 -16674.852,E2 -16674.852} C_VEL
LIN {X 0,Y 291.42,Z 309.088,A -85,B 0,C 180,E1 -16677.466,E2 -16677.466} C_VEL
LIN {X 0,Y 291.315,Z 309.004,A -85,B 0,C 180,E1 -16680.439,E2 -16680.439} C_VEL
LIN {X 0,Y 291.341,Z 309.002,A -85,B 0,C 180,E1 -16683.698,E2 -16683.698} C_VEL
LIN {X 0,Y 291.355,Z 309.006,A -85,B 0,C 180,E1 -16687.249,E2 -16687.249} C_VEL
LIN {X 0,Y 291.295,Z 309,A -85,B 0,C 180,E1 -16690.648,E2 -16690.648} C_VEL
LIN {X 0,Y 291.277,Z 309.011,A -85,B 0,C 180,E1 -16694.403,E2 -16694.403} C_VEL
LIN {X 0,Y 291.289,Z 309.007,A -85,B 0,C 180,E1 -16698.411,E2 -16698.411} C_VEL
LIN {X 0,Y 291.327,Z 308.986,A -85,B 0,C 180,E1 -16701.154,E2 -16701.154} C_VEL
LIN {X 0,Y 291.349,Z 309.001,A -85,B 0,C 180,E1 -16704.625,E2 -16704.625} C_VEL
LIN {X 0,Y 291.36,Z 309.002,A -85,B 0,C 180,E1 -16707.949,E2 -16707.949} C_VEL
LIN {X 0,Y 291.336,Z 309.004,A -85,B 0,C 180,E1 -16711.153,E2 -16711.153} C_VEL
LIN {X 0,Y 291.335,Z 309.007,A -85,B 0,C 180,E1 -16714.264,E2 -16714.264} C_VEL
LIN {X 0,Y 291.342,Z 308.996,A -85,B 0,C 180,E1 -16717.296,E2 -16717.296} C_VEL
LIN {X 0,Y 291.378,Z 309,A -85,B 0,C 180,E1 -16720.265,E2 -16720.265} C_VEL
LIN {X 0,Y 291.467,Z 308.984,A -85,B 0,C 180,E1 -16724.682,E2 -16724.682} C_VEL
LIN {X 0,Y 291.519,Z 308.982,A -85,B 0,C 180,E1 -16728.88,E2 -16728.88} C_VEL
LIN {X 0,Y 291.644,Z 308.967,A -85,B 0,C 180,E1 -16731.687,E2 -16731.687} C_VEL
LIN {X 0,Y 291.588,Z 308.965,A -85,B 0,C 180,E1 -16734.468,E2 -16734.468} C_VEL
LIN {X 0,Y 291.861,Z 308.94,A -85,B 0,C 180,E1 -16738.62,E2 -16738.62} C_VEL
LIN {X 0,Y 291.86,Z 308.94,A -85,B 0,C 180,E1 -16741.38,E2 -16741.38} C_VEL
LIN {X 0,Y 291.676,Z 308.959,A -85,B 0,C 180,E1 -16746.92,E2 -16746.92} C_VEL
LIN {X 0,Y 291.556,Z 308.982,A -85,B 0,C 180,E1 -16749.715,E2 -16749.715} C_VEL
LIN {X 0,Y 291.473,Z 308.981,A -85,B 0,C 180,E1 -16753.953,E2 -16753.953} C_VEL
LIN {X 0,Y 291.397,Z 308.996,A -85,B 0,C 180,E1 -16756.823,E2 -16756.823} C_VEL
LIN {X 0,Y 291.385,Z 308.998,A -85,B 0,C 180,E1 -16759.843,E2 -16759.843} C_VEL
LIN {X 0,Y 291.319,Z 309.006,A -85,B 0,C 180,E1 -16764.213,E2 -16764.213} C_VEL
LIN {X 0,Y 291.343,Z 309.008,A -85,B 0,C 180,E1 -16767.28,E2 -16767.28} C_VEL
LIN {X 0,Y 291.312,Z 309.002,A -85,B 0,C 180,E1 -16770.44,E2 -16770.44} C_VEL
LIN {X 0,Y 291.338,Z 309.006,A -85,B 0,C 180,E1 -16773.699,E2 -16773.699} C_VEL
LIN {X 0,Y 291.343,Z 308.991,A -85,B 0,C 180,E1 -16777.247,E2 -16777.247} C_VEL
LIN {X 0,Y 291.295,Z 308.995,A -85,B 0,C 180,E1 -16780.649,E2 -16780.649} C_VEL
LIN {X 0,Y 291.278,Z 309.014,A -85,B 0,C 180,E1 -16784.405,E2 -16784.405} C_VEL
LIN {X 0,Y 291.29,Z 308.998,A -85,B 0,C 180,E1 -16788.413,E2 -16788.413} C_VEL
LIN {X 0,Y 291.331,Z 309.008,A -85,B 0,C 180,E1 -16791.156,E2 -16791.156} C_VEL
LIN {X 0,Y 291.353,Z 308.998,A -85,B 0,C 180,E1 -16794.626,E2 -16794.626} C_VEL
LIN {X 0,Y 291.364,Z 309.004,A -85,B 0,C 180,E1 -16797.951,E2 -16797.951} C_VEL
LIN {X 0,Y 291.376,Z 309.086,A -85,B 0,C 180,E1 -16802.53,E2 -16802.53} C_VEL
LIN {X 0,Y 292.972,Z 317.166,A -85,B 0,C 180,E1 -16805.933,E2 -16805.933} C_VEL
LIN {X 0,Y 293.493,Z 321.069,A -85,B 0,C 180,E1 -16807.472,E2 -16807.472} C_VEL
LIN {X 0,Y 293.517,Z 323.839,A -85,B 0,C 180,E1 -16808.412,E2 -16808.412} C_VEL
LIN {X 0,Y 295.109,Z 331.701,A -85,B 0,C 180,E1 -16808.79,E2 -16808.79} C_VEL
LIN {X 0,Y 299.159,Z 355.703,A -85,B 0,C 180,E1 -16809.695,E2 -16809.695} C_VEL
LIN {X 0,Y 298.247,Z 400.048,A -85,B 0,C 180,E1 -16810.782,E2 -16810.782} C_VEL
LIN {X 0,Y 297.81,Z 409.825,A -85,B 0,C 180,E1 -16811.2,E2 -16811.2} C_VEL
LIN {X 0,Y 297.046,Z 420.912,A -85,B 0,C 180,E1 -16811.909,E2 -16811.909} C_VEL
LIN {X 0,Y 295.984,Z 431.732,A -85,B 0,C 180,E1 -16812.913,E2 -16812.913} C_VEL
LIN {X 0,Y 294.97,Z 440.131,A -85,B 0,C 180,E1 -16813.92,E2 -16813.92} C_VEL
LIN {X 0,Y 293.925,Z 448.063,A -85,B 0,C 180,E1 -16815.106,E2 -16815.106} C_VEL
LIN {X 0,Y 292.934,Z 455.46,A -85,B 0,C 180,E1 -16816.472,E2 -16816.472} C_VEL
LIN {X 0,Y 291.787,Z 462.955,A -85,B 0,C 180,E1 -16818.187,E2 -16818.187} C_VEL
LIN {X 0,Y 290.824,Z 469.828,A -85,B 0,C 180,E1 -16820.261,E2 -16820.261} C_VEL
LIN {X 0,Y 290.117,Z 475.024,A -85,B 0,C 180,E1 -16822.344,E2 -16822.344} C_VEL
LIN {X 0,Y 289.748,Z 478.093,A -85,B 0,C 180,E1 -16823.978,E2 -16823.978} C_VEL
LIN {X 0,Y 289.556,Z 480.612,A -85,B 0,C 180,E1 -16825.824,E2 -16825.824} C_VEL
LIN {X 0,Y 289.465,Z 481.887,A -85,B 0,C 180,E1 -16827.217,E2 -16827.217} C_VEL
LIN {X 0,Y 289.385,Z 482.692,A -85,B 0,C 180,E1 -16828.608,E2 -16828.608} C_VEL
LIN {X 0,Y 289.352,Z 482.998,A -85,B 0,C 180,E1 -16830,E2 -16830} C_VEL
LIN {X 0,Y 289.381,Z 482.719,A -85,B 0,C 180,E1 -16831.392,E2 -16831.392} C_VEL
LIN {X 0,Y 289.453,Z 481.968,A -85,B 0,C 180,E1 -16832.783,E2 -16832.783} C_VEL
LIN {X 0,Y 289.535,Z 480.747,A -85,B 0,C 180,E1 -16834.176,E2 -16834.176} C_VEL
LIN {X 0,Y 289.754,Z 478.265,A -85,B 0,C 180,E1 -16836.033,E2 -16836.033} C_VEL
LIN {X 0,Y 290.112,Z 475.275,A -85,B 0,C 180,E1 -16837.657,E2 -16837.657} C_VEL
LIN {X 0,Y 290.76,Z 470.147,A -85,B 0,C 180,E1 -16839.741,E2 -16839.741} C_VEL
LIN {X 0,Y 291.559,Z 464.631,A -85,B 0,C 180,E1 -16841.47,E2 -16841.47} C_VEL
LIN {X 0,Y 292.638,Z 457.702,A -85,B 0,C 180,E1 -16843.188,E2 -16843.188} C_VEL
LIN {X 0,Y 293.707,Z 449.748,A -85,B 0,C 180,E1 -16844.728,E2 -16844.728} C_VEL
LIN {X 0,Y 294.77,Z 442.165,A -85,B 0,C 180,E1 -16845.913,E2 -16845.913} C_VEL
LIN {X 0,Y 295.754,Z 434.216,A -85,B 0,C 180,E1 -16846.923,E2 -16846.923} C_VEL
LIN {X 0,Y 296.587,Z 426.005,A -85,B 0,C 180,E1 -16847.763,E2 -16847.763} C_VEL
LIN {X 0,Y 297.354,Z 417.681,A -85,B 0,C 180,E1 -16848.428,E2 -16848.428} C_VEL
LIN {X 0,Y 297.87,Z 408.676,A -85,B 0,C 180,E1 -16848.975,E2 -16848.975} C_VEL
LIN {X 0,Y 298.324,Z 398.872,A -85,B 0,C 180,E1 -16849.37,E2 -16849.37} C_VEL
LIN {X 0,Y 299.16,Z 355.432,A -85,B 0,C 180,E1 -16850.43,E2 -16850.43} C_VEL
LIN {X 0,Y 295.325,Z 332.766,A -85,B 0,C 180,E1 -16851.285,E2 -16851.285} C_VEL
LIN {X 0,Y 293.557,Z 323.879,A -85,B 0,C 180,E1 -16851.698,E2 -16851.698} C_VEL
LIN {X 0,Y 293.508,Z 321.383,A -85,B 0,C 180,E1 -16852.526,E2 -16852.526} C_VEL
LIN {X 0,Y 292.685,Z 315.522,A -85,B 0,C 180,E1 -16854.849,E2 -16854.849} C_VEL
LIN {X 0,Y 291.435,Z 309.082,A -85,B 0,C 180,E1 -16857.561,E2 -16857.561} C_VEL
LIN {X 0,Y 291.364,Z 309.004,A -85,B 0,C 180,E1 -16862.049,E2 -16862.049} C_VEL
LIN {X 0,Y 291.353,Z 308.998,A -85,B 0,C 180,E1 -16865.374,E2 -16865.374} C_VEL
LIN {X 0,Y 291.331,Z 309.008,A -85,B 0,C 180,E1 -16868.844,E2 -16868.844} C_VEL
LIN {X 0,Y 291.283,Z 309.001,A -85,B 0,C 180,E1 -16872.498,E2 -16872.498} C_VEL
LIN {X 0,Y 291.285,Z 309.012,A -85,B 0,C 180,E1 -16876.37,E2 -16876.37} C_VEL
LIN {X 0,Y 291.307,Z 308.99,A -85,B 0,C 180,E1 -16880.534,E2 -16880.534} C_VEL
LIN {X 0,Y 291.381,Z 308.987,A -85,B 0,C 180,E1 -16882.915,E2 -16882.915} C_VEL
LIN {X 0,Y 291.338,Z 309.005,A -85,B 0,C 180,E1 -16886.301,E2 -16886.301} C_VEL
LIN {X 0,Y 291.359,Z 308.998,A -85,B 0,C 180,E1 -16890.268,E2 -16890.268} C_VEL
LIN {X 0,Y 291.328,Z 309.007,A -85,B 0,C 180,E1 -16894.378,E2 -16894.378} C_VEL
LIN {X 0,Y 290.621,Z 309.094,A -85,B 0,C 180,E1 -16895.532,E2 -16895.532} C_VEL
LIN {X 0,Y 287.787,Z 309.439,A -85,B 0,C 180,E1 -16897.413,E2 -16897.413} C_VEL
LIN {X 0,Y 285.409,Z 309.741,A -85,B 0,C 180,E1 -16898.94,E2 -16898.94} C_VEL
LIN {X 0,Y 284.387,Z 309.869,A -85,B 0,C 180,E1 -16900.122,E2 -16900.122} C_VEL
LIN {X 0,Y 284.302,Z 309.877,A -85,B 0,C 180,E1 -16900.522,E2 -16900.522} C_VEL
LIN {X 0,Y 284.408,Z 309.865,A -85,B 0,C 180,E1 -16904.516,E2 -16904.516} C_VEL
LIN {X 0,Y 284.452,Z 309.864,A -85,B 0,C 180,E1 -16908.6,E2 -16908.6} C_VEL
LIN {X 0,Y 284.601,Z 309.844,A -85,B 0,C 180,E1 -16911.479,E2 -16911.479} C_VEL
LIN {X 0,Y 284.559,Z 309.841,A -85,B 0,C 180,E1 -16914.33,E2 -16914.33} C_VEL
LIN {X 0,Y 284.829,Z 309.816,A -85,B 0,C 180,E1 -16918.586,E2 -16918.586} C_VEL
LIN {X 0,Y 284.827,Z 309.816,A -85,B 0,C 180,E1 -16921.414,E2 -16921.414} C_VEL
LIN {X 0,Y 284.629,Z 309.837,A -85,B 0,C 180,E1 -16927.092,E2 -16927.092} C_VEL
LIN {X 0,Y 284.503,Z 309.858,A -85,B 0,C 180,E1 -16929.957,E2 -16929.957} C_VEL
LIN {X 0,Y 284.41,Z 309.861,A -85,B 0,C 180,E1 -16934.306,E2 -16934.306} C_VEL
LIN {X 0,Y 284.342,Z 309.877,A -85,B 0,C 180,E1 -16937.253,E2 -16937.253} C_VEL
LIN {X 0,Y 284.315,Z 309.876,A -85,B 0,C 180,E1 -16940.247,E2 -16940.247} C_VEL
LIN {X 0,Y 284.286,Z 309.883,A -85,B 0,C 180,E1 -16943.84,E2 -16943.84} C_VEL
LIN {X 0,Y 284.274,Z 309.882,A -85,B 0,C 180,E1 -16948.017,E2 -16948.017} C_VEL
LIN {X 0,Y 284.279,Z 309.884,A -85,B 0,C 180,E1 -16951.276,E2 -16951.276} C_VEL
LIN {X 0,Y 284.33,Z 309.874,A -85,B 0,C 180,E1 -16955.347,E2 -16955.347} C_VEL
LIN {X 0,Y 284.287,Z 309.864,A -85,B 0,C 180,E1 -16958.173,E2 -16958.173} C_VEL
LIN {X 0,Y 284.231,Z 309.886,A -85,B 0,C 180,E1 -16962.117,E2 -16962.117} C_VEL
LIN {X 0,Y 284.232,Z 309.888,A -85,B 0,C 180,E1 -16966.186,E2 -16966.186} C_VEL
LIN {X 0,Y 284.279,Z 309.877,A -85,B 0,C 180,E1 -16970.03,E2 -16970.03} C_VEL
LIN {X 0,Y 284.318,Z 309.878,A -85,B 0,C 180,E1 -16973.613,E2 -16973.613} C_VEL
LIN {X 0,Y 284.303,Z 309.884,A -85,B 0,C 180,E1 -16977.191,E2 -16977.191} C_VEL
LIN {X 0,Y 284.334,Z 309.879,A -85,B 0,C 180,E1 -16980.374,E2 -16980.374} C_VEL
LIN {X 0,Y 284.406,Z 310.138,A -85,B 0,C 180,E1 -16982.23,E2 -16982.23} C_VEL
LIN {X 0,Y 286.177,Z 319.51,A -85,B 0,C 180,E1 -16986.173,E2 -16986.173} C_VEL
LIN {X 0,Y 286.621,Z 323.784,A -85,B 0,C 180,E1 -16987.781,E2 -16987.781} C_VEL
LIN {X 0,Y 287.848,Z 329.469,A -85,B 0,C 180,E1 -16988.093,E2 -16988.093} C_VEL
LIN {X 0,Y 291.354,Z 348.747,A -85,B 0,C 180,E1 -16988.87,E2 -16988.87} C_VEL
LIN {X 0,Y 292.569,Z 358.048,A -85,B 0,C 180,E1 -16989.202,E2 -16989.202} C_VEL
LIN {X 0,Y 291.671,Z 399.995,A -85,B 0,C 180,E1 -16990.255,E2 -16990.255} C_VEL
LIN {X 0,Y 291.152,Z 409.511,A -85,B 0,C 180,E1 -16990.662,E2 -16990.662} C_VEL
LIN {X 0,Y 290.412,Z 419.497,A -85,B 0,C 180,E1 -16991.298,E2 -16991.298} C_VEL
LIN {X 0,Y 289.343,Z 430.841,A -85,B 0,C 180,E1 -16992.325,E2 -16992.325} C_VEL
LIN {X 0,Y 288.319,Z 439.399,A -85,B 0,C 180,E1 -16993.357,E2 -16993.357} C_VEL
LIN {X 0,Y 287.166,Z 447.451,A -85,B 0,C 180,E1 -16994.565,E2 -16994.565} C_VEL
LIN {X 0,Y 286.205,Z 454.101,A -85,B 0,C 180,E1 -16995.786,E2 -16995.786} C_VEL
LIN {X 0,Y 285.266,Z 460.412,A -85,B 0,C 180,E1 -16997.19,E2 -16997.19} C_VEL
LIN {X 0,Y 284.424,Z 465.655,A -85,B 0,C 180,E1 -16998.599,E2 -16998.599} C_VEL
LIN {X 0,Y 283.774,Z 470.026,A -85,B 0,C 180,E1 -17000.017,E2 -17000.017} C_VEL
LIN {X 0,Y 283.063,Z 475.179,A -85,B 0,C 180,E1 -17002.152,E2 -17002.152} C_VEL
LIN {X 0,Y 282.61,Z 478.96,A -85,B 0,C 180,E1 -17004.291,E2 -17004.291} C_VEL
LIN {X 0,Y 282.461,Z 480.695,A -85,B 0,C 180,E1 -17005.719,E2 -17005.719} C_VEL
LIN {X 0,Y 282.374,Z 481.937,A -85,B 0,C 180,E1 -17007.147,E2 -17007.147} C_VEL
LIN {X 0,Y 282.309,Z 482.709,A -85,B 0,C 180,E1 -17008.574,E2 -17008.574} C_VEL
LIN {X 0,Y 282.274,Z 483,A -85,B 0,C 180,E1 -17010,E2 -17010} C_VEL
LIN {X 0,Y 282.309,Z 482.702,A -85,B 0,C 180,E1 -17011.426,E2 -17011.426} C_VEL
LIN {X 0,Y 282.374,Z 481.918,A -85,B 0,C 180,E1 -17012.853,E2 -17012.853} C_VEL
LIN {X 0,Y 282.459,Z 480.663,A -85,B 0,C 180,E1 -17014.281,E2 -17014.281} C_VEL
LIN {X 0,Y 282.638,Z 478.54,A -85,B 0,C 180,E1 -17015.942,E2 -17015.942} C_VEL
LIN {X 0,Y 283.063,Z 475.12,A -85,B 0,C 180,E1 -17017.848,E2 -17017.848} C_VEL
LIN {X 0,Y 283.77,Z 469.949,A -85,B 0,C 180,E1 -17019.983,E2 -17019.983} C_VEL
LIN {X 0,Y 284.831,Z 463.13,A -85,B 0,C 180,E1 -17022.106,E2 -17022.106} C_VEL
LIN {X 0,Y 285.975,Z 455.674,A -85,B 0,C 180,E1 -17023.863,E2 -17023.863} C_VEL
LIN {X 0,Y 287.033,Z 448.319,A -85,B 0,C 180,E1 -17025.26,E2 -17025.26} C_VEL
LIN {X 0,Y 288.139,Z 440.439,A -85,B 0,C 180,E1 -17026.471,E2 -17026.471} C_VEL
LIN {X 0,Y 289.173,Z 432.107,A -85,B 0,C 180,E1 -17027.503,E2 -17027.503} C_VEL
LIN {X 0,Y 290.221,Z 421.452,A -85,B 0,C 180,E1 -17028.532,E2 -17028.532} C_VEL
LIN {X 0,Y 291.048,Z 410.653,A -85,B 0,C 180,E1 -17029.254,E2 -17029.254} C_VEL
LIN {X 0,Y 291.55,Z 401.339,A -85,B 0,C 180,E1 -17029.677,E2 -17029.677} C_VEL
LIN {X 0,Y 292.12,Z 375.867,A -85,B 0,C 180,E1 -17030.344,E2 -17030.344} C_VEL
LIN {X 0,Y 292.465,Z 356.38,A -85,B 0,C 180,E1 -17030.82,E2 -17030.82} C_VEL
LIN {X 0,Y 288.794,Z 334.416,A -85,B 0,C 180,E1 -17031.671,E2 -17031.671} C_VEL
LIN {X 0,Y 286.63,Z 324.086,A -85,B 0,C 180,E1 -17032.148,E2 -17032.148} C_VEL
LIN {X 0,Y 286.535,Z 322.988,A -85,B 0,C 180,E1 -17032.42,E2 -17032.42} C_VEL
LIN {X 0,Y 285.791,Z 317.281,A -85,B 0,C 180,E1 -17034.711,E2 -17034.711} C_VEL
LIN {X 0,Y 284.377,Z 309.95,A -85,B 0,C 180,E1 -17037.889,E2 -17037.889} C_VEL
LIN {X 0,Y 284.282,Z 309.881,A -85,B 0,C 180,E1 -17041.275,E2 -17041.275} C_VEL
LIN {X 0,Y 284.333,Z 309.871,A -85,B 0,C 180,E1 -17045.346,E2 -17045.346} C_VEL
LIN {X 0,Y 284.294,Z 309.883,A -85,B 0,C 180,E1 -17048.171,E2 -17048.171} C_VEL
LIN {X 0,Y 284.231,Z 309.878,A -85,B 0,C 180,E1 -17052.116,E2 -17052.116} C_VEL
LIN {X 0,Y 284.232,Z 309.891,A -85,B 0,C 180,E1 -17056.185,E2 -17056.185} C_VEL
LIN {X 0,Y 284.278,Z 309.865,A -85,B 0,C 180,E1 -17060.029,E2 -17060.029} C_VEL
LIN {X 0,Y 284.312,Z 309.874,A -85,B 0,C 180,E1 -17063.611,E2 -17063.611} C_VEL
LIN {X 0,Y 284.3,Z 309.883,A -85,B 0,C 180,E1 -17067.19,E2 -17067.19} C_VEL
LIN {X 0,Y 284.33,Z 309.872,A -85,B 0,C 180,E1 -17070.373,E2 -17070.373} C_VEL
LIN {X 0,Y 284.29,Z 309.883,A -85,B 0,C 180,E1 -17073.578,E2 -17073.578} C_VEL
LIN {X 0,Y 284.301,Z 309.876,A -85,B 0,C 180,E1 -17076.701,E2 -17076.701} C_VEL
LIN {X 0,Y 284.327,Z 309.875,A -85,B 0,C 180,E1 -17079.928,E2 -17079.928} C_VEL
LIN {X 0,Y 284.408,Z 309.864,A -85,B 0,C 180,E1 -17084.516,E2 -17084.516} C_VEL
LIN {X 0,Y 284.451,Z 309.864,A -85,B 0,C 180,E1 -17088.6,E2 -17088.6} C_VEL
LIN {X 0,Y 284.601,Z 309.844,A -85,B 0,C 180,E1 -17091.48,E2 -17091.48} C_VEL
LIN {X 0,Y 284.558,Z 309.84,A -85,B 0,C 180,E1 -17094.331,E2 -17094.331} C_VEL
LIN {X 0,Y 284.829,Z 309.816,A -85,B 0,C 180,E1 -17098.586,E2 -17098.586} C_VEL
LIN {X 0,Y 284.827,Z 309.816,A -85,B 0,C 180,E1 -17101.414,E2 -17101.414} C_VEL
LIN {X 0,Y 284.629,Z 309.837,A -85,B 0,C 180,E1 -17107.092,E2 -17107.092} C_VEL
LIN {X 0,Y 284.503,Z 309.858,A -85,B 0,C 180,E1 -17109.958,E2 -17109.958} C_VEL
LIN {X 0,Y 284.411,Z 309.86,A -85,B 0,C 180,E1 -17114.307,E2 -17114.307} C_VEL
LIN {X 0,Y 284.342,Z 309.877,A -85,B 0,C 180,E1 -17117.254,E2 -17117.254} C_VEL
LIN {X 0,Y 284.316,Z 309.876,A -85,B 0,C 180,E1 -17120.247,E2 -17120.247} C_VEL
LIN {X 0,Y 284.287,Z 309.883,A -85,B 0,C 180,E1 -17123.84,E2 -17123.84} C_VEL
LIN {X 0,Y 284.274,Z 309.882,A -85,B 0,C 180,E1 -17128.017,E2 -17128.017} C_VEL
LIN {X 0,Y 284.279,Z 309.883,A -85,B 0,C 180,E1 -17131.276,E2 -17131.276} C_VEL
LIN {X 0,Y 284.331,Z 309.875,A -85,B 0,C 180,E1 -17135.347,E2 -17135.347} C_VEL
LIN {X 0,Y 284.288,Z 309.865,A -85,B 0,C 180,E1 -17138.173,E2 -17138.173} C_VEL
LIN {X 0,Y 284.232,Z 309.885,A -85,B 0,C 180,E1 -17142.118,E2 -17142.118} C_VEL
LIN {X 0,Y 284.234,Z 309.889,A -85,B 0,C 180,E1 -17146.186,E2 -17146.186} C_VEL
LIN {X 0,Y 284.281,Z 309.876,A -85,B 0,C 180,E1 -17150.031,E2 -17150.031} C_VEL
LIN {X 0,Y 284.319,Z 309.878,A -85,B 0,C 180,E1 -17153.613,E2 -17153.613} C_VEL
LIN {X 0,Y 284.304,Z 309.884,A -85,B 0,C 180,E1 -17157.191,E2 -17157.191} C_VEL
LIN {X 0,Y 284.347,Z 309.901,A -85,B 0,C 180,E1 -17161.992,E2 -17161.992} C_VEL
LIN {X 0,Y 284.443,Z 310.521,A -85,B 0,C 180,E1 -17162.477,E2 -17162.477} C_VEL
LIN {X 0,Y 285.864,Z 317.574,A -85,B 0,C 180,E1 -17165.457,E2 -17165.457} C_VEL
LIN {X 0,Y 286.532,Z 322.85,A -85,B 0,C 180,E1 -17167.58,E2 -17167.58} C_VEL
LIN {X 0,Y 286.627,Z 324.145,A -85,B 0,C 180,E1 -17167.903,E2 -17167.903} C_VEL
LIN {X 0,Y 289.94,Z 340.328,A -85,B 0,C 180,E1 -17168.618,E2 -17168.618} C_VEL
LIN {X 0,Y 292.507,Z 356.887,A -85,B 0,C 180,E1 -17169.242,E2 -17169.242} C_VEL
LIN {X 0,Y 291.559,Z 400.066,A -85,B 0,C 180,E1 -17170.324,E2 -17170.324} C_VEL
LIN {X 0,Y 291.109,Z 409.836,A -85,B 0,C 180,E1 -17170.75,E2 -17170.75} C_VEL
LIN {X 0,Y 290.315,Z 420.919,A -85,B 0,C 180,E1 -17171.475,E2 -17171.475} C_VEL
LIN {X 0,Y 289.224,Z 431.737,A -85,B 0,C 180,E1 -17172.5,E2 -17172.5} C_VEL
LIN {X 0,Y 288.169,Z 440.135,A -85,B 0,C 180,E1 -17173.53,E2 -17173.53} C_VEL
LIN {X 0,Y 287.073,Z 448.066,A -85,B 0,C 180,E1 -17174.742,E2 -17174.742} C_VEL
LIN {X 0,Y 286.034,Z 455.463,A -85,B 0,C 180,E1 -17176.14,E2 -17176.14} C_VEL
LIN {X 0,Y 284.849,Z 462.957,A -85,B 0,C 180,E1 -17177.894,E2 -17177.894} C_VEL
LIN {X 0,Y 283.823,Z 469.83,A -85,B 0,C 180,E1 -17180.019,E2 -17180.019} C_VEL
LIN {X 0,Y 283.07,Z 475.025,A -85,B 0,C 180,E1 -17182.152,E2 -17182.152} C_VEL
LIN {X 0,Y 282.639,Z 478.467,A -85,B 0,C 180,E1 -17184.058,E2 -17184.058} C_VEL
LIN {X 0,Y 282.465,Z 480.613,A -85,B 0,C 180,E1 -17185.719,E2 -17185.719} C_VEL
LIN {X 0,Y 282.377,Z 481.888,A -85,B 0,C 180,E1 -17187.147,E2 -17187.147} C_VEL
LIN {X 0,Y 282.311,Z 482.692,A -85,B 0,C 180,E1 -17188.574,E2 -17188.574} C_VEL
LIN {X 0,Y 282.276,Z 482.998,A -85,B 0,C 180,E1 -17190,E2 -17190} C_VEL
LIN {X 0,Y 282.307,Z 482.719,A -85,B 0,C 180,E1 -17191.426,E2 -17191.426} C_VEL
LIN {X 0,Y 282.364,Z 481.967,A -85,B 0,C 180,E1 -17192.853,E2 -17192.853} C_VEL
LIN {X 0,Y 282.446,Z 480.746,A -85,B 0,C 180,E1 -17194.281,E2 -17194.281} C_VEL
LIN {X 0,Y 282.641,Z 478.652,A -85,B 0,C 180,E1 -17195.945,E2 -17195.945} C_VEL
LIN {X 0,Y 283.064,Z 475.274,A -85,B 0,C 180,E1 -17197.848,E2 -17197.848} C_VEL
LIN {X 0,Y 283.745,Z 470.145,A -85,B 0,C 180,E1 -17199.984,E2 -17199.984} C_VEL
LIN {X 0,Y 284.6,Z 464.629,A -85,B 0,C 180,E1 -17201.755,E2 -17201.755} C_VEL
LIN {X 0,Y 285.737,Z 457.699,A -85,B 0,C 180,E1 -17203.512,E2 -17203.512} C_VEL
LIN {X 0,Y 286.856,Z 449.744,A -85,B 0,C 180,E1 -17205.088,E2 -17205.088} C_VEL
LIN {X 0,Y 287.959,Z 442.16,A -85,B 0,C 180,E1 -17206.3,E2 -17206.3} C_VEL
LIN {X 0,Y 288.971,Z 434.211,A -85,B 0,C 180,E1 -17207.333,E2 -17207.333} C_VEL
LIN {X 0,Y 289.845,Z 425.999,A -85,B 0,C 180,E1 -17208.191,E2 -17208.191} C_VEL
LIN {X 0,Y 290.643,Z 417.673,A -85,B 0,C 180,E1 -17208.869,E2 -17208.869} C_VEL
LIN {X 0,Y 291.169,Z 408.665,A -85,B 0,C 180,E1 -17209.429,E2 -17209.429} C_VEL
LIN {X 0,Y 291.601,Z 399.747,A -85,B 0,C 180,E1 -17209.804,E2 -17209.804} C_VEL
LIN {X 0,Y 292.435,Z 355.917,A -85,B 0,C 180,E1 -17210.908,E2 -17210.908} C_VEL
LIN {X 0,Y 288.919,Z 334.792,A -85,B 0,C 180,E1 -17211.727,E2 -17211.727} C_VEL
LIN {X 0,Y 286.633,Z 324.004,A -85,B 0,C 180,E1 -17212.238,E2 -17212.238} C_VEL
LIN {X 0,Y 286.527,Z 322.356,A -85,B 0,C 180,E1 -17212.725,E2 -17212.725} C_VEL
LIN {X 0,Y 285.467,Z 315.524,A -85,B 0,C 180,E1 -17215.52,E2 -17215.52} C_VEL
LIN {X 0,Y 284.367,Z 309.966,A -85,B 0,C 180,E1 -17217.949,E2 -17217.949} C_VEL
LIN {X 0,Y 284.283,Z 309.88,A -85,B 0,C 180,E1 -17221.275,E2 -17221.275} C_VEL
LIN {X 0,Y 284.335,Z 309.871,A -85,B 0,C 180,E1 -17225.346,E2 -17225.346} C_VEL
LIN {X 0,Y 284.295,Z 309.883,A -85,B 0,C 180,E1 -17228.171,E2 -17228.171} C_VEL
LIN {X 0,Y 284.232,Z 309.877,A -85,B 0,C 180,E1 -17232.116,E2 -17232.116} C_VEL
LIN {X 0,Y 284.233,Z 309.891,A -85,B 0,C 180,E1 -17236.185,E2 -17236.185} C_VEL
LIN {X 0,Y 284.251,Z 309.87,A -85,B 0,C 180,E1 -17240.036,E2 -17240.036} C_VEL
LIN {X 0,Y 284.314,Z 309.874,A -85,B 0,C 180,E1 -17243.611,E2 -17243.611} C_VEL
LIN {X 0,Y 284.301,Z 309.884,A -85,B 0,C 180,E1 -17247.19,E2 -17247.19} C_VEL
LIN {X 0,Y 284.331,Z 309.873,A -85,B 0,C 180,E1 -17250.373,E2 -17250.373} C_VEL
LIN {X 0,Y 284.257,Z 309.884,A -85,B 0,C 180,E1 -17254.376,E2 -17254.376} C_VEL
LIN {X 0,Y 284.291,Z 309.875,A -85,B 0,C 180,E1 -17258.234,E2 -17258.234} C_VEL
LIN {X 0,Y 284.302,Z 309.877,A -85,B 0,C 180,E1 -17260.522,E2 -17260.522} C_VEL
LIN {X 0,Y 283.645,Z 309.964,A -85,B 0,C 180,E1 -17261.705,E2 -17261.705} C_VEL
LIN {X 0,Y 280.863,Z 310.31,A -85,B 0,C 180,E1 -17263.635,E2 -17263.635} C_VEL
LIN {X 0,Y 278.495,Z 310.603,A -85,B 0,C 180,E1 -17265.202,E2 -17265.202} C_VEL
LIN {X 0,Y 277.461,Z 310.727,A -85,B 0,C 180,E1 -17266.415,E2 -17266.415} C_VEL
LIN {X 0,Y 277.367,Z 310.737,A -85,B 0,C 180,E1 -17266.825,E2 -17266.825} C_VEL
LIN {X 0,Y 277.564,Z 310.72,A -85,B 0,C 180,E1 -17271.262,E2 -17271.262} C_VEL
LIN {X 0,Y 277.529,Z 310.716,A -85,B 0,C 180,E1 -17274.186,E2 -17274.186} C_VEL
LIN {X 0,Y 277.796,Z 310.693,A -85,B 0,C 180,E1 -17278.55,E2 -17278.55} C_VEL
LIN {X 0,Y 277.794,Z 310.693,A -85,B 0,C 180,E1 -17281.45,E2 -17281.45} C_VEL
LIN {X 0,Y 277.585,Z 310.715,A -85,B 0,C 180,E1 -17287.273,E2 -17287.273} C_VEL
LIN {X 0,Y 277.444,Z 310.735,A -85,B 0,C 180,E1 -17290.213,E2 -17290.213} C_VEL
LIN {X 0,Y 277.363,Z 310.737,A -85,B 0,C 180,E1 -17294.678,E2 -17294.678} C_VEL
LIN {X 0,Y 277.27,Z 310.76,A -85,B 0,C 180,E1 -17299.239,E2 -17299.239} C_VEL
LIN {X 0,Y 277.249,Z 310.759,A -85,B 0,C 180,E1 -17303.928,E2 -17303.928} C_VEL
LIN {X 0,Y 277.26,Z 310.759,A -85,B 0,C 180,E1 -17307.482,E2 -17307.482} C_VEL
LIN {X 0,Y 277.243,Z 310.755,A -85,B 0,C 180,E1 -17310.473,E2 -17310.473} C_VEL
LIN {X 0,Y 277.24,Z 310.761,A -85,B 0,C 180,E1 -17313.896,E2 -17313.896} C_VEL
LIN {X 0,Y 277.242,Z 310.742,A -85,B 0,C 180,E1 -17317.473,E2 -17317.473} C_VEL
LIN {X 0,Y 277.178,Z 310.758,A -85,B 0,C 180,E1 -17321.242,E2 -17321.242} C_VEL
LIN {X 0,Y 277.169,Z 310.77,A -85,B 0,C 180,E1 -17325.233,E2 -17325.233} C_VEL
LIN {X 0,Y 277.179,Z 310.752,A -85,B 0,C 180,E1 -17328.759,E2 -17328.759} C_VEL
LIN {X 0,Y 277.251,Z 310.764,A -85,B 0,C 180,E1 -17332.529,E2 -17332.529} C_VEL
LIN {X 0,Y 277.243,Z 310.757,A -85,B 0,C 180,E1 -17336.105,E2 -17336.105} C_VEL
LIN {X 0,Y 277.26,Z 310.754,A -85,B 0,C 180,E1 -17339.539,E2 -17339.539} C_VEL
LIN {X 0,Y 277.338,Z 310.982,A -85,B 0,C 180,E1 -17341.81,E2 -17341.81} C_VEL
LIN {X 0,Y 279.077,Z 319.954,A -85,B 0,C 180,E1 -17345.708,E2 -17345.708} C_VEL
LIN {X 0,Y 279.623,Z 323.798,A -85,B 0,C 180,E1 -17347.195,E2 -17347.195} C_VEL
LIN {X 0,Y 281.155,Z 329.937,A -85,B 0,C 180,E1 -17347.556,E2 -17347.556} C_VEL
LIN {X 0,Y 284.766,Z 349.718,A -85,B 0,C 180,E1 -17348.383,E2 -17348.383} C_VEL
LIN {X 0,Y 285.892,Z 357.164,A -85,B 0,C 180,E1 -17348.669,E2 -17348.669} C_VEL
LIN {X 0,Y 285.002,Z 399.845,A -85,B 0,C 180,E1 -17349.767,E2 -17349.767} C_VEL
LIN {X 0,Y 284.472,Z 409.521,A -85,B 0,C 180,E1 -17350.189,E2 -17350.189} C_VEL
LIN {X 0,Y 283.71,Z 419.504,A -85,B 0,C 180,E1 -17350.839,E2 -17350.839} C_VEL
LIN {X 0,Y 282.584,Z 430.845,A -85,B 0,C 180,E1 -17351.888,E2 -17351.888} C_VEL
LIN {X 0,Y 281.522,Z 439.403,A -85,B 0,C 180,E1 -17352.943,E2 -17352.943} C_VEL
LIN {X 0,Y 280.341,Z 447.454,A -85,B 0,C 180,E1 -17354.18,E2 -17354.18} C_VEL
LIN {X 0,Y 279.318,Z 454.103,A -85,B 0,C 180,E1 -17355.427,E2 -17355.427} C_VEL
LIN {X 0,Y 278.356,Z 460.414,A -85,B 0,C 180,E1 -17356.866,E2 -17356.866} C_VEL
LIN {X 0,Y 277.461,Z 465.657,A -85,B 0,C 180,E1 -17358.309,E2 -17358.309} C_VEL
LIN {X 0,Y 276.78,Z 470.027,A -85,B 0,C 180,E1 -17359.762,E2 -17359.762} C_VEL
LIN {X 0,Y 276.039,Z 475.18,A -85,B 0,C 180,E1 -17361.951,E2 -17361.951} C_VEL
LIN {X 0,Y 275.549,Z 478.961,A -85,B 0,C 180,E1 -17364.145,E2 -17364.145} C_VEL
LIN {X 0,Y 275.374,Z 480.696,A -85,B 0,C 180,E1 -17365.609,E2 -17365.609} C_VEL
LIN {X 0,Y 275.288,Z 481.938,A -85,B 0,C 180,E1 -17367.073,E2 -17367.073} C_VEL
LIN {X 0,Y 275.237,Z 482.709,A -85,B 0,C 180,E1 -17368.537,E2 -17368.537} C_VEL
LIN {X 0,Y 275.2,Z 483,A -85,B 0,C 180,E1 -17370,E2 -17370} C_VEL
LIN {X 0,Y 275.237,Z 482.702,A -85,B 0,C 180,E1 -17371.463,E2 -17371.463} C_VEL
LIN {X 0,Y 275.288,Z 481.918,A -85,B 0,C 180,E1 -17372.927,E2 -17372.927} C_VEL
LIN {X 0,Y 275.372,Z 480.663,A -85,B 0,C 180,E1 -17374.391,E2 -17374.391} C_VEL
LIN {X 0,Y 275.672,Z 477.763,A -85,B 0,C 180,E1 -17376.588,E2 -17376.588} C_VEL
LIN {X 0,Y 276.038,Z 475.119,A -85,B 0,C 180,E1 -17378.049,E2 -17378.049} C_VEL
LIN {X 0,Y 276.774,Z 469.948,A -85,B 0,C 180,E1 -17380.238,E2 -17380.238} C_VEL
LIN {X 0,Y 277.9,Z 463.128,A -85,B 0,C 180,E1 -17382.413,E2 -17382.413} C_VEL
LIN {X 0,Y 279.075,Z 455.672,A -85,B 0,C 180,E1 -17384.213,E2 -17384.213} C_VEL
LIN {X 0,Y 280.196,Z 448.316,A -85,B 0,C 180,E1 -17385.642,E2 -17385.642} C_VEL
LIN {X 0,Y 281.346,Z 440.435,A -85,B 0,C 180,E1 -17386.881,E2 -17386.881} C_VEL
LIN {X 0,Y 282.396,Z 432.102,A -85,B 0,C 180,E1 -17387.937,E2 -17387.937} C_VEL
LIN {X 0,Y 283.513,Z 421.445,A -85,B 0,C 180,E1 -17388.987,E2 -17388.987} C_VEL
LIN {X 0,Y 284.366,Z 410.644,A -85,B 0,C 180,E1 -17389.725,E2 -17389.725} C_VEL
LIN {X 0,Y 284.89,Z 401.324,A -85,B 0,C 180,E1 -17390.157,E2 -17390.157} C_VEL
LIN {X 0,Y 285.48,Z 375.673,A -85,B 0,C 180,E1 -17390.844,E2 -17390.844} C_VEL
LIN {X 0,Y 285.764,Z 356.649,A -85,B 0,C 180,E1 -17391.324,E2 -17391.324} C_VEL
LIN {X 0,Y 282.059,Z 334.626,A -85,B 0,C 180,E1 -17392.209,E2 -17392.209} C_VEL
LIN {X 0,Y 279.84,Z 325.001,A -85,B 0,C 180,E1 -17392.669,E2 -17392.669} C_VEL
LIN {X 0,Y 279.541,Z 323.504,A -85,B 0,C 180,E1 -17392.847,E2 -17392.847} C_VEL
LIN {X 0,Y 278.575,Z 317.279,A -85,B 0,C 180,E1 -17395.396,E2 -17395.396} C_VEL
LIN {X 0,Y 277.311,Z 310.839,A -85,B 0,C 180,E1 -17398.277,E2 -17398.277} C_VEL
LIN {X 0,Y 277.237,Z 310.764,A -85,B 0,C 180,E1 -17402.164,E2 -17402.164} C_VEL
LIN {X 0,Y 277.271,Z 310.754,A -85,B 0,C 180,E1 -17405.796,E2 -17405.796} C_VEL
LIN {X 0,Y 277.213,Z 310.76,A -85,B 0,C 180,E1 -17409.331,E2 -17409.331} C_VEL
LIN {X 0,Y 277.186,Z 310.76,A -85,B 0,C 180,E1 -17413.201,E2 -17413.201} C_VEL
LIN {X 0,Y 277.187,Z 310.765,A -85,B 0,C 180,E1 -17417.33,E2 -17417.33} C_VEL
LIN {X 0,Y 277.244,Z 310.739,A -85,B 0,C 180,E1 -17421.796,E2 -17421.796} C_VEL
LIN {X 0,Y 277.271,Z 310.751,A -85,B 0,C 180,E1 -17424.34,E2 -17424.34} C_VEL
LIN {X 0,Y 277.234,Z 310.762,A -85,B 0,C 180,E1 -17427.835,E2 -17427.835} C_VEL
LIN {X 0,Y 277.232,Z 310.76,A -85,B 0,C 180,E1 -17431.206,E2 -17431.206} C_VEL
LIN {X 0,Y 277.225,Z 310.767,A -85,B 0,C 180,E1 -17434.471,E2 -17434.471} C_VEL
LIN {X 0,Y 277.24,Z 310.751,A -85,B 0,C 180,E1 -17437.651,E2 -17437.651} C_VEL
LIN {X 0,Y 277.27,Z 310.76,A -85,B 0,C 180,E1 -17440.761,E2 -17440.761} C_VEL
LIN {X 0,Y 277.364,Z 310.737,A -85,B 0,C 180,E1 -17445.322,E2 -17445.322} C_VEL
LIN {X 0,Y 277.447,Z 310.735,A -85,B 0,C 180,E1 -17449.787,E2 -17449.787} C_VEL
LIN {X 0,Y 277.593,Z 310.714,A -85,B 0,C 180,E1 -17452.728,E2 -17452.728} C_VEL
LIN {X 0,Y 277.796,Z 310.693,A -85,B 0,C 180,E1 -17458.55,E2 -17458.55} C_VEL
LIN {X 0,Y 277.794,Z 310.693,A -85,B 0,C 180,E1 -17461.45,E2 -17461.45} C_VEL
LIN {X 0,Y 277.585,Z 310.715,A -85,B 0,C 180,E1 -17467.273,E2 -17467.273} C_VEL
LIN {X 0,Y 277.444,Z 310.735,A -85,B 0,C 180,E1 -17470.214,E2 -17470.214} C_VEL
LIN {X 0,Y 277.364,Z 310.737,A -85,B 0,C 180,E1 -17474.678,E2 -17474.678} C_VEL
LIN {X 0,Y 277.27,Z 310.76,A -85,B 0,C 180,E1 -17479.239,E2 -17479.239} C_VEL
LIN {X 0,Y 277.249,Z 310.759,A -85,B 0,C 180,E1 -17483.928,E2 -17483.928} C_VEL
LIN {X 0,Y 277.261,Z 310.759,A -85,B 0,C 180,E1 -17487.482,E2 -17487.482} C_VEL
LIN {X 0,Y 277.243,Z 310.754,A -85,B 0,C 180,E1 -17490.473,E2 -17490.473} C_VEL
LIN {X 0,Y 277.241,Z 310.761,A -85,B 0,C 180,E1 -17493.897,E2 -17493.897} C_VEL
LIN {X 0,Y 277.243,Z 310.743,A -85,B 0,C 180,E1 -17497.473,E2 -17497.473} C_VEL
LIN {X 0,Y 277.179,Z 310.756,A -85,B 0,C 180,E1 -17501.242,E2 -17501.242} C_VEL
LIN {X 0,Y 277.17,Z 310.77,A -85,B 0,C 180,E1 -17505.233,E2 -17505.233} C_VEL
LIN {X 0,Y 277.18,Z 310.752,A -85,B 0,C 180,E1 -17508.759,E2 -17508.759} C_VEL
LIN {X 0,Y 277.253,Z 310.763,A -85,B 0,C 180,E1 -17512.529,E2 -17512.529} C_VEL
LIN {X 0,Y 277.244,Z 310.756,A -85,B 0,C 180,E1 -17516.105,E2 -17516.105} C_VEL
LIN {X 0,Y 277.227,Z 310.759,A -85,B 0,C 180,E1 -17519.535,E2 -17519.535} C_VEL
LIN {X 0,Y 277.33,Z 311.014,A -85,B 0,C 180,E1 -17521.909,E2 -17521.909} C_VEL
LIN {X 0,Y 279.044,Z 319.765,A -85,B 0,C 180,E1 -17525.707,E2 -17525.707} C_VEL
LIN {X 0,Y 279.582,Z 323.845,A -85,B 0,C 180,E1 -17527.277,E2 -17527.277} C_VEL
LIN {X 0,Y 281.325,Z 330.912,A -85,B 0,C 180,E1 -17527.674,E2 -17527.674} C_VEL
LIN {X 0,Y 284.891,Z 350.957,A -85,B 0,C 180,E1 -17528.502,E2 -17528.502} C_VEL
LIN {X 0,Y 285.864,Z 357.704,A -85,B 0,C 180,E1 -17528.757,E2 -17528.757} C_VEL
LIN {X 0,Y 284.904,Z 400.083,A -85,B 0,C 180,E1 -17529.844,E2 -17529.844} C_VEL
LIN {X 0,Y 284.426,Z 409.847,A -85,B 0,C 180,E1 -17530.28,E2 -17530.28} C_VEL
LIN {X 0,Y 283.59,Z 420.927,A -85,B 0,C 180,E1 -17531.019,E2 -17531.019} C_VEL
LIN {X 0,Y 282.475,Z 431.742,A -85,B 0,C 180,E1 -17532.068,E2 -17532.068} C_VEL
LIN {X 0,Y 281.375,Z 440.139,A -85,B 0,C 180,E1 -17533.121,E2 -17533.121} C_VEL
LIN {X 0,Y 280.239,Z 448.07,A -85,B 0,C 180,E1 -17534.36,E2 -17534.36} C_VEL
LIN {X 0,Y 279.116,Z 455.466,A -85,B 0,C 180,E1 -17535.789,E2 -17535.789} C_VEL
LIN {X 0,Y 277.918,Z 462.959,A -85,B 0,C 180,E1 -17537.588,E2 -17537.588} C_VEL
LIN {X 0,Y 276.815,Z 469.832,A -85,B 0,C 180,E1 -17539.763,E2 -17539.763} C_VEL
LIN {X 0,Y 276.045,Z 475.026,A -85,B 0,C 180,E1 -17541.951,E2 -17541.951} C_VEL
LIN {X 0,Y 275.674,Z 477.693,A -85,B 0,C 180,E1 -17543.413,E2 -17543.413} C_VEL
LIN {X 0,Y 275.377,Z 480.613,A -85,B 0,C 180,E1 -17545.609,E2 -17545.609} C_VEL
LIN {X 0,Y 275.291,Z 481.888,A -85,B 0,C 180,E1 -17547.073,E2 -17547.073} C_VEL
LIN {X 0,Y 275.238,Z 482.692,A -85,B 0,C 180,E1 -17548.537,E2 -17548.537} C_VEL
LIN {X 0,Y 275.201,Z 482.998,A -85,B 0,C 180,E1 -17550,E2 -17550} C_VEL
LIN {X 0,Y 275.234,Z 482.719,A -85,B 0,C 180,E1 -17551.463,E2 -17551.463} C_VEL
LIN {X 0,Y 275.279,Z 481.967,A -85,B 0,C 180,E1 -17552.927,E2 -17552.927} C_VEL
LIN {X 0,Y 275.36,Z 480.745,A -85,B 0,C 180,E1 -17554.391,E2 -17554.391} C_VEL
LIN {X 0,Y 275.674,Z 477.88,A -85,B 0,C 180,E1 -17556.587,E2 -17556.587} C_VEL
LIN {X 0,Y 276.038,Z 475.272,A -85,B 0,C 180,E1 -17558.049,E2 -17558.049} C_VEL
LIN {X 0,Y 276.753,Z 470.144,A -85,B 0,C 180,E1 -17560.239,E2 -17560.239} C_VEL
LIN {X 0,Y 277.659,Z 464.627,A -85,B 0,C 180,E1 -17562.053,E2 -17562.053} C_VEL
LIN {X 0,Y 278.833,Z 457.697,A -85,B 0,C 180,E1 -17563.854,E2 -17563.854} C_VEL
LIN {X 0,Y 279.996,Z 449.741,A -85,B 0,C 180,E1 -17565.467,E2 -17565.467} C_VEL
LIN {X 0,Y 281.164,Z 442.156,A -85,B 0,C 180,E1 -17566.705,E2 -17566.705} C_VEL
LIN {X 0,Y 282.218,Z 434.206,A -85,B 0,C 180,E1 -17567.761,E2 -17567.761} C_VEL
LIN {X 0,Y 283.119,Z 425.993,A -85,B 0,C 180,E1 -17568.638,E2 -17568.638} C_VEL
LIN {X 0,Y 283.928,Z 417.731,A -85,B 0,C 180,E1 -17569.328,E2 -17569.328} C_VEL
LIN {X 0,Y 284.471,Z 408.845,A -85,B 0,C 180,E1 -17569.894,E2 -17569.894} C_VEL
LIN {X 0,Y 284.946,Z 399.909,A -85,B 0,C 180,E1 -17570.28,E2 -17570.28} C_VEL
LIN {X 0,Y 285.797,Z 356.484,A -85,B 0,C 180,E1 -17571.402,E2 -17571.402} C_VEL
LIN {X 0,Y 282.01,Z 334.259,A -85,B 0,C 180,E1 -17572.301,E2 -17572.301} C_VEL
LIN {X 0,Y 279.829,Z 324.877,A -85,B 0,C 180,E1 -17572.753,E2 -17572.753} C_VEL
LIN {X 0,Y 279.561,Z 323.451,A -85,B 0,C 180,E1 -17572.934,E2 -17572.934} C_VEL
LIN {X 0,Y 278.623,Z 317.474,A -85,B 0,C 180,E1 -17575.391,E2 -17575.391} C_VEL
LIN {X 0,Y 277.32,Z 310.846,A -85,B 0,C 180,E1 -17578.363,E2 -17578.363} C_VEL
LIN {X 0,Y 277.238,Z 310.764,A -85,B 0,C 180,E1 -17582.164,E2 -17582.164} C_VEL
LIN {X 0,Y 277.272,Z 310.752,A -85,B 0,C 180,E1 -17585.796,E2 -17585.796} C_VEL
LIN {X 0,Y 277.214,Z 310.761,A -85,B 0,C 180,E1 -17589.33,E2 -17589.33} C_VEL
LIN {X 0,Y 277.187,Z 310.759,A -85,B 0,C 180,E1 -17593.201,E2 -17593.201} C_VEL
LIN {X 0,Y 277.188,Z 310.766,A -85,B 0,C 180,E1 -17597.33,E2 -17597.33} C_VEL
LIN {X 0,Y 277.218,Z 310.741,A -85,B 0,C 180,E1 -17601.803,E2 -17601.803} C_VEL
LIN {X 0,Y 277.272,Z 310.75,A -85,B 0,C 180,E1 -17604.339,E2 -17604.339} C_VEL
LIN {X 0,Y 277.235,Z 310.762,A -85,B 0,C 180,E1 -17607.835,E2 -17607.835} C_VEL
LIN {X 0,Y 277.232,Z 310.759,A -85,B 0,C 180,E1 -17611.206,E2 -17611.206} C_VEL
LIN {X 0,Y 277.226,Z 310.766,A -85,B 0,C 180,E1 -17614.471,E2 -17614.471} C_VEL
LIN {X 0,Y 277.241,Z 310.751,A -85,B 0,C 180,E1 -17617.651,E2 -17617.651} C_VEL
LIN {X 0,Y 277.27,Z 310.76,A -85,B 0,C 180,E1 -17620.761,E2 -17620.761} C_VEL
LIN {X 0,Y 277.364,Z 310.737,A -85,B 0,C 180,E1 -17625.322,E2 -17625.322} C_VEL
LIN {X 0,Y 277.367,Z 310.737,A -85,B 0,C 180,E1 -17626.825,E2 -17626.825} C_VEL
LIN {X 0,Y 276.699,Z 310.824,A -85,B 0,C 180,E1 -17628.039,E2 -17628.039} C_VEL
LIN {X 0,Y 273.943,Z 311.173,A -85,B 0,C 180,E1 -17630.021,E2 -17630.021} C_VEL
LIN {X 0,Y 271.61,Z 311.463,A -85,B 0,C 180,E1 -17631.631,E2 -17631.631} C_VEL
LIN {X 0,Y 270.595,Z 311.585,A -85,B 0,C 180,E1 -17632.875,E2 -17632.875} C_VEL
LIN {X 0,Y 270.504,Z 311.592,A -85,B 0,C 180,E1 -17633.297,E2 -17633.297} C_VEL
LIN {X 0,Y 270.761,Z 311.569,A -85,B 0,C 180,E1 -17638.512,E2 -17638.512} C_VEL
LIN {X 0,Y 270.76,Z 311.569,A -85,B 0,C 180,E1 -17641.487,E2 -17641.487} C_VEL
LIN {X 0,Y 270.545,Z 311.592,A -85,B 0,C 180,E1 -17647.463,E2 -17647.463} C_VEL
LIN {X 0,Y 270.377,Z 311.615,A -85,B 0,C 180,E1 -17650.483,E2 -17650.483} C_VEL
LIN {X 0,Y 270.331,Z 311.614,A -85,B 0,C 180,E1 -17655.069,E2 -17655.069} C_VEL
LIN {X 0,Y 270.213,Z 311.635,A -85,B 0,C 180,E1 -17659.762,E2 -17659.762} C_VEL
LIN {X 0,Y 270.176,Z 311.639,A -85,B 0,C 180,E1 -17664.436,E2 -17664.436} C_VEL
LIN {X 0,Y 270.19,Z 311.636,A -85,B 0,C 180,E1 -17667.918,E2 -17667.918} C_VEL
LIN {X 0,Y 270.168,Z 311.641,A -85,B 0,C 180,E1 -17671.35,E2 -17671.35} C_VEL
LIN {X 0,Y 270.191,Z 311.639,A -85,B 0,C 180,E1 -17674.907,E2 -17674.907} C_VEL
LIN {X 0,Y 270.193,Z 311.611,A -85,B 0,C 180,E1 -17678.711,E2 -17678.711} C_VEL
LIN {X 0,Y 270.143,Z 311.648,A -85,B 0,C 180,E1 -17683.245,E2 -17683.245} C_VEL
LIN {X 0,Y 270.146,Z 311.631,A -85,B 0,C 180,E1 -17687.438,E2 -17687.438} C_VEL
LIN {X 0,Y 270.204,Z 311.639,A -85,B 0,C 180,E1 -17691.375,E2 -17691.375} C_VEL
LIN {X 0,Y 270.195,Z 311.629,A -85,B 0,C 180,E1 -17695.094,E2 -17695.094} C_VEL
LIN {X 0,Y 270.182,Z 311.635,A -85,B 0,C 180,E1 -17699.137,E2 -17699.137} C_VEL
LIN {X 0,Y 270.279,Z 311.812,A -85,B 0,C 180,E1 -17701.354,E2 -17701.354} C_VEL
LIN {X 0,Y 272.114,Z 321.27,A -85,B 0,C 180,E1 -17705.592,E2 -17705.592} C_VEL
LIN {X 0,Y 272.533,Z 323.795,A -85,B 0,C 180,E1 -17706.566,E2 -17706.566} C_VEL
LIN {X 0,Y 274.393,Z 330.125,A -85,B 0,C 180,E1 -17706.976,E2 -17706.976} C_VEL
LIN {X 0,Y 278.193,Z 350.853,A -85,B 0,C 180,E1 -17707.875,E2 -17707.875} C_VEL
LIN {X 0,Y 279.298,Z 358.605,A -85,B 0,C 180,E1 -17708.178,E2 -17708.178} C_VEL
LIN {X 0,Y 278.365,Z 399.985,A -85,B 0,C 180,E1 -17709.267,E2 -17709.267} C_VEL
LIN {X 0,Y 277.818,Z 409.53,A -85,B 0,C 180,E1 -17709.694,E2 -17709.694} C_VEL
LIN {X 0,Y 276.942,Z 420.71,A -85,B 0,C 180,E1 -17710.449,E2 -17710.449} C_VEL
LIN {X 0,Y 275.848,Z 430.849,A -85,B 0,C 180,E1 -17711.43,E2 -17711.43} C_VEL
LIN {X 0,Y 274.74,Z 439.406,A -85,B 0,C 180,E1 -17712.509,E2 -17712.509} C_VEL
LIN {X 0,Y 273.523,Z 447.457,A -85,B 0,C 180,E1 -17713.774,E2 -17713.774} C_VEL
LIN {X 0,Y 272.442,Z 454.106,A -85,B 0,C 180,E1 -17715.051,E2 -17715.051} C_VEL
LIN {X 0,Y 271.44,Z 460.417,A -85,B 0,C 180,E1 -17716.525,E2 -17716.525} C_VEL
LIN {X 0,Y 270.518,Z 465.659,A -85,B 0,C 180,E1 -17718.005,E2 -17718.005} C_VEL
LIN {X 0,Y 269.803,Z 470.029,A -85,B 0,C 180,E1 -17719.494,E2 -17719.494} C_VEL
LIN {X 0,Y 268.994,Z 475.181,A -85,B 0,C 180,E1 -17721.738,E2 -17721.738} C_VEL
LIN {X 0,Y 268.499,Z 478.962,A -85,B 0,C 180,E1 -17723.99,E2 -17723.99} C_VEL
LIN {X 0,Y 268.291,Z 480.696,A -85,B 0,C 180,E1 -17725.493,E2 -17725.493} C_VEL
LIN {X 0,Y 268.205,Z 481.938,A -85,B 0,C 180,E1 -17726.996,E2 -17726.996} C_VEL
LIN {X 0,Y 268.144,Z 482.709,A -85,B 0,C 180,E1 -17728.498,E2 -17728.498} C_VEL
LIN {X 0,Y 268.128,Z 483,A -85,B 0,C 180,E1 -17730,E2 -17730} C_VEL
LIN {X 0,Y 268.144,Z 482.702,A -85,B 0,C 180,E1 -17731.502,E2 -17731.502} C_VEL
LIN {X 0,Y 268.204,Z 481.918,A -85,B 0,C 180,E1 -17733.004,E2 -17733.004} C_VEL
LIN {X 0,Y 268.409,Z 479.306,A -85,B 0,C 180,E1 -17735.739,E2 -17735.739} C_VEL
LIN {X 0,Y 268.801,Z 476.594,A -85,B 0,C 180,E1 -17737.512,E2 -17737.512} C_VEL
LIN {X 0,Y 269.483,Z 471.859,A -85,B 0,C 180,E1 -17739.76,E2 -17739.76} C_VEL
LIN {X 0,Y 270.304,Z 466.729,A -85,B 0,C 180,E1 -17741.625,E2 -17741.625} C_VEL
LIN {X 0,Y 271.178,Z 461.713,A -85,B 0,C 180,E1 -17743.107,E2 -17743.107} C_VEL
LIN {X 0,Y 272.193,Z 455.669,A -85,B 0,C 180,E1 -17744.58,E2 -17744.58} C_VEL
LIN {X 0,Y 273.375,Z 448.313,A -85,B 0,C 180,E1 -17746.043,E2 -17746.043} C_VEL
LIN {X 0,Y 274.566,Z 440.431,A -85,B 0,C 180,E1 -17747.311,E2 -17747.311} C_VEL
LIN {X 0,Y 275.669,Z 432.098,A -85,B 0,C 180,E1 -17748.39,E2 -17748.39} C_VEL
LIN {X 0,Y 276.825,Z 421.439,A -85,B 0,C 180,E1 -17749.464,E2 -17749.464} C_VEL
LIN {X 0,Y 277.746,Z 409.802,A -85,B 0,C 180,E1 -17750.263,E2 -17750.263} C_VEL
LIN {X 0,Y 278.266,Z 401.141,A -85,B 0,C 180,E1 -17750.664,E2 -17750.664} C_VEL
LIN {X 0,Y 278.999,Z 370.053,A -85,B 0,C 180,E1 -17751.503,E2 -17751.503} C_VEL
LIN {X 0,Y 279.172,Z 357.598,A -85,B 0,C 180,E1 -17751.826,E2 -17751.826} C_VEL
LIN {X 0,Y 275.189,Z 334.01,A -85,B 0,C 180,E1 -17752.811,E2 -17752.811} C_VEL
LIN {X 0,Y 273.198,Z 326.194,A -85,B 0,C 180,E1 -17753.205,E2 -17753.205} C_VEL
LIN {X 0,Y 272.488,Z 323.674,A -85,B 0,C 180,E1 -17753.43,E2 -17753.43} C_VEL
LIN {X 0,Y 271.347,Z 317.277,A -85,B 0,C 180,E1 -17756.123,E2 -17756.123} C_VEL
LIN {X 0,Y 270.268,Z 311.723,A -85,B 0,C 180,E1 -17758.695,E2 -17758.695} C_VEL
LIN {X 0,Y 270.212,Z 311.633,A -85,B 0,C 180,E1 -17763.665,E2 -17763.665} C_VEL
LIN {X 0,Y 270.206,Z 311.636,A -85,B 0,C 180,E1 -17766.742,E2 -17766.742} C_VEL
LIN {X 0,Y 270.143,Z 311.63,A -85,B 0,C 180,E1 -17770.57,E2 -17770.57} C_VEL
LIN {X 0,Y 270.124,Z 311.647,A -85,B 0,C 180,E1 -17774.625,E2 -17774.625} C_VEL
LIN {X 0,Y 270.146,Z 311.641,A -85,B 0,C 180,E1 -17777.437,E2 -17777.437} C_VEL
LIN {X 0,Y 270.187,Z 311.612,A -85,B 0,C 180,E1 -17781.371,E2 -17781.371} C_VEL
LIN {X 0,Y 270.192,Z 311.639,A -85,B 0,C 180,E1 -17785.093,E2 -17785.093} C_VEL
LIN {X 0,Y 270.179,Z 311.635,A -85,B 0,C 180,E1 -17789.136,E2 -17789.136} C_VEL
LIN {X 0,Y 270.193,Z 311.637,A -85,B 0,C 180,E1 -17792.172,E2 -17792.172} C_VEL
LIN {X 0,Y 270.176,Z 311.639,A -85,B 0,C 180,E1 -17795.564,E2 -17795.564} C_VEL
LIN {X 0,Y 270.213,Z 311.635,A -85,B 0,C 180,E1 -17800.238,E2 -17800.238} C_VEL
LIN {X 0,Y 270.331,Z 311.613,A -85,B 0,C 180,E1 -17804.931,E2 -17804.931} C_VEL
LIN {X 0,Y 270.379,Z 311.614,A -85,B 0,C 180,E1 -17809.517,E2 -17809.517} C_VEL
LIN {X 0,Y 270.555,Z 311.591,A -85,B 0,C 180,E1 -17812.537,E2 -17812.537} C_VEL
LIN {X 0,Y 270.761,Z 311.569,A -85,B 0,C 180,E1 -17818.513,E2 -17818.513} C_VEL
LIN {X 0,Y 270.76,Z 311.569,A -85,B 0,C 180,E1 -17821.488,E2 -17821.488} C_VEL
LIN {X 0,Y 270.546,Z 311.592,A -85,B 0,C 180,E1 -17827.463,E2 -17827.463} C_VEL
LIN {X 0,Y 270.377,Z 311.615,A -85,B 0,C 180,E1 -17830.484,E2 -17830.484} C_VEL
LIN {X 0,Y 270.331,Z 311.613,A -85,B 0,C 180,E1 -17835.069,E2 -17835.069} C_VEL
LIN {X 0,Y 270.213,Z 311.635,A -85,B 0,C 180,E1 -17839.762,E2 -17839.762} C_VEL
LIN {X 0,Y 270.176,Z 311.639,A -85,B 0,C 180,E1 -17844.436,E2 -17844.436} C_VEL
LIN {X 0,Y 270.19,Z 311.637,A -85,B 0,C 180,E1 -17847.918,E2 -17847.918} C_VEL
LIN {X 0,Y 270.169,Z 311.64,A -85,B 0,C 180,E1 -17851.35,E2 -17851.35} C_VEL
LIN {X 0,Y 270.192,Z 311.639,A -85,B 0,C 180,E1 -17854.907,E2 -17854.907} C_VEL
LIN {X 0,Y 270.194,Z 311.611,A -85,B 0,C 180,E1 -17858.711,E2 -17858.711} C_VEL
LIN {X 0,Y 270.144,Z 311.647,A -85,B 0,C 180,E1 -17863.246,E2 -17863.246} C_VEL
LIN {X 0,Y 270.147,Z 311.632,A -85,B 0,C 180,E1 -17867.438,E2 -17867.438} C_VEL
LIN {X 0,Y 270.205,Z 311.639,A -85,B 0,C 180,E1 -17871.375,E2 -17871.375} C_VEL
LIN {X 0,Y 270.196,Z 311.629,A -85,B 0,C 180,E1 -17875.095,E2 -17875.095} C_VEL
LIN {X 0,Y 270.17,Z 311.637,A -85,B 0,C 180,E1 -17879.142,E2 -17879.142} C_VEL
LIN {X 0,Y 270.257,Z 311.845,A -85,B 0,C 180,E1 -17881.457,E2 -17881.457} C_VEL
LIN {X 0,Y 272.094,Z 321.074,A -85,B 0,C 180,E1 -17885.59,E2 -17885.59} C_VEL
LIN {X 0,Y 272.557,Z 323.889,A -85,B 0,C 180,E1 -17886.663,E2 -17886.663} C_VEL
LIN {X 0,Y 274.63,Z 331.417,A -85,B 0,C 180,E1 -17887.113,E2 -17887.113} C_VEL
LIN {X 0,Y 278.082,Z 350.38,A -85,B 0,C 180,E1 -17887.932,E2 -17887.932} C_VEL
LIN {X 0,Y 279.233,Z 359.091,A -85,B 0,C 180,E1 -17888.264,E2 -17888.264} C_VEL
LIN {X 0,Y 278.242,Z 400.364,A -85,B 0,C 180,E1 -17889.35,E2 -17889.35} C_VEL
LIN {X 0,Y 277.705,Z 410.69,A -85,B 0,C 180,E1 -17889.83,E2 -17889.83} C_VEL
LIN {X 0,Y 276.66,Z 422.926,A -85,B 0,C 180,E1 -17890.717,E2 -17890.717} C_VEL
LIN {X 0,Y 275.743,Z 431.747,A -85,B 0,C 180,E1 -17891.615,E2 -17891.615} C_VEL
LIN {X 0,Y 274.588,Z 440.143,A -85,B 0,C 180,E1 -17892.691,E2 -17892.691} C_VEL
LIN {X 0,Y 273.421,Z 448.073,A -85,B 0,C 180,E1 -17893.96,E2 -17893.96} C_VEL
LIN {X 0,Y 272.226,Z 455.469,A -85,B 0,C 180,E1 -17895.421,E2 -17895.421} C_VEL
LIN {X 0,Y 270.975,Z 462.962,A -85,B 0,C 180,E1 -17897.265,E2 -17897.265} C_VEL
LIN {X 0,Y 269.831,Z 469.833,A -85,B 0,C 180,E1 -17899.495,E2 -17899.495} C_VEL
LIN {X 0,Y 269,Z 475.028,A -85,B 0,C 180,E1 -17901.738,E2 -17901.738} C_VEL
LIN {X 0,Y 268.62,Z 477.694,A -85,B 0,C 180,E1 -17903.239,E2 -17903.239} C_VEL
LIN {X 0,Y 268.411,Z 479.243,A -85,B 0,C 180,E1 -17904.259,E2 -17904.259} C_VEL
LIN {X 0,Y 268.207,Z 481.889,A -85,B 0,C 180,E1 -17906.996,E2 -17906.996} C_VEL
LIN {X 0,Y 268.146,Z 482.692,A -85,B 0,C 180,E1 -17908.498,E2 -17908.498} C_VEL
LIN {X 0,Y 268.129,Z 482.998,A -85,B 0,C 180,E1 -17910,E2 -17910} C_VEL
LIN {X 0,Y 268.141,Z 482.718,A -85,B 0,C 180,E1 -17911.502,E2 -17911.502} C_VEL
LIN {X 0,Y 268.195,Z 481.967,A -85,B 0,C 180,E1 -17913.004,E2 -17913.004} C_VEL
LIN {X 0,Y 268.407,Z 479.412,A -85,B 0,C 180,E1 -17915.733,E2 -17915.733} C_VEL
LIN {X 0,Y 268.802,Z 476.722,A -85,B 0,C 180,E1 -17917.511,E2 -17917.511} C_VEL
LIN {X 0,Y 269.461,Z 472.053,A -85,B 0,C 180,E1 -17919.76,E2 -17919.76} C_VEL
LIN {X 0,Y 270.304,Z 466.969,A -85,B 0,C 180,E1 -17921.625,E2 -17921.625} C_VEL
LIN {X 0,Y 271.175,Z 462.003,A -85,B 0,C 180,E1 -17923.107,E2 -17923.107} C_VEL
LIN {X 0,Y 272.147,Z 456.01,A -85,B 0,C 180,E1 -17924.583,E2 -17924.583} C_VEL
LIN {X 0,Y 273.307,Z 448.717,A -85,B 0,C 180,E1 -17926.047,E2 -17926.047} C_VEL
LIN {X 0,Y 274.555,Z 440.923,A -85,B 0,C 180,E1 -17927.312,E2 -17927.312} C_VEL
LIN {X 0,Y 275.683,Z 432.701,A -85,B 0,C 180,E1 -17928.389,E2 -17928.389} C_VEL
LIN {X 0,Y 276.605,Z 424.114,A -85,B 0,C 180,E1 -17929.287,E2 -17929.287} C_VEL
LIN {X 0,Y 277.554,Z 413.588,A -85,B 0,C 180,E1 -17930.119,E2 -17930.119} C_VEL
LIN {X 0,Y 278.268,Z 402.096,A -85,B 0,C 180,E1 -17930.706,E2 -17930.706} C_VEL
LIN {X 0,Y 278.702,Z 383.349,A -85,B 0,C 180,E1 -17931.244,E2 -17931.244} C_VEL
LIN {X 0,Y 279.292,Z 358.067,A -85,B 0,C 180,E1 -17931.882,E2 -17931.882} C_VEL
LIN {X 0,Y 275.791,Z 337.067,A -85,B 0,C 180,E1 -17932.754,E2 -17932.754} C_VEL
LIN {X 0,Y 273.466,Z 326.901,A -85,B 0,C 180,E1 -17933.242,E2 -17933.242} C_VEL
LIN {X 0,Y 272.468,Z 323.634,A -85,B 0,C 180,E1 -17933.514,E2 -17933.514} C_VEL
LIN {X 0,Y 271.379,Z 317.473,A -85,B 0,C 180,E1 -17936.119,E2 -17936.119} C_VEL
LIN {X 0,Y 270.26,Z 311.74,A -85,B 0,C 180,E1 -17938.755,E2 -17938.755} C_VEL
LIN {X 0,Y 270.213,Z 311.634,A -85,B 0,C 180,E1 -17943.665,E2 -17943.665} C_VEL
LIN {X 0,Y 270.207,Z 311.636,A -85,B 0,C 180,E1 -17946.742,E2 -17946.742} C_VEL
LIN {X 0,Y 270.144,Z 311.631,A -85,B 0,C 180,E1 -17950.57,E2 -17950.57} C_VEL
